(* check if inputs have chaged and fill buffer *)
IF s0 <> X0 THEN
	esr_out[cnt].typ := 10 + BOOL_TO_BYTE(s0);
	esr_out[cnt].adress := a0;
	esr_out[cnt].DS := DT_in;
	esr_out[cnt].TS := TX;
	X0 := S0;
	cnt := cnt + 1;
	esr_flag := TRUE;
END_IF;
IF s1 <> X1 THEN
	esr_out[cnt].typ := 10 + BOOL_TO_BYTE(s1);
	esr_out[cnt].adress := a1;
	esr_out[cnt].DS := DT_in;
	esr_out[cnt].TS := TX;
	X1 := S1;
	cnt := cnt + 1;
	esr_flag := TRUE;
END_IF;
IF s2 <> X2 THEN
	esr_out[cnt].typ := 10 + BOOL_TO_BYTE(s2);
	esr_out[cnt].adress := a2;
	esr_out[cnt].DS := DT_in;
	esr_out[cnt].TS := TX;
	X2 := S2;
	cnt := cnt + 1;
	esr_flag := TRUE;
END_IF;
IF s3 <> X3 THEN
	esr_out[cnt].typ := 10 + BOOL_TO_BYTE(s3);
	esr_out[cnt].adress := a3;
	esr_out[cnt].DS := DT_in;
	esr_out[cnt].TS := TX;
	X3 := S3;
	cnt := cnt + 1;
	esr_flag := TRUE;
END_IF;
IF s4 <> X4 AND cnt < 4 THEN
	esr_out[cnt].typ := 10 + BOOL_TO_BYTE(s4);
	esr_out[cnt].adress := a4;
	esr_out[cnt].DS := DT_in;
	esr_out[cnt].TS := TX;
	X4 := S4;
	cnt := cnt + 1;
	esr_flag := TRUE;
END_IF;
IF s5 <> X5  AND cnt < 4 THEN
	esr_out[cnt].typ := 10 + BOOL_TO_BYTE(s5);
	esr_out[cnt].adress := a5;
	esr_out[cnt].DS := DT_in;
	esr_out[cnt].TS := TX;
	X5 := S5;
	cnt := cnt + 1;
	esr_flag := TRUE;
END_IF;
IF s6 <> X6  AND cnt < 4 THEN
	esr_out[cnt].typ := 10 + BOOL_TO_BYTE(s6);
	esr_out[cnt].adress := a6;
	esr_out[cnt].DS := DT_in;
	esr_out[cnt].TS := TX;
	X6 := S6;
	cnt := cnt + 1;
	esr_flag := TRUE;
END_IF;
IF s7 <> X7  AND cnt < 4 THEN
	esr_out[cnt].typ := 10 + BOOL_TO_BYTE(s7);
	esr_out[cnt].adress := a7;
	esr_out[cnt].DS := DT_in;
	esr_out[cnt].TS := TX;
	X7 := S7;
	cnt := cnt + 1;
	esr_flag := TRUE;
END_IF;

(* revision history
hm	26. jan 2007	rev 1.0
	original version

hm	17. sep 2007	rev 1.1
	replaced time() with T_PLC_MS() for compatibility reasons

hm	22. oct. 2008	rev 1.2
	optimized code

hm	1.dec. 2009	rev 1.3
	changed esr_out to be I/O

*)
END_FUNCTION_BLOCK

(* POU Other/ESR_MON_R4, ST *)
FUNCTION_BLOCK ESR_MON_R4
VAR_INPUT
	R0, R1, R2, R3 : REAL;
	DT_in : DT;
END_VAR
VAR_INPUT CONSTANT
	a0, a1, a2, a3 : STRING(10);
	s0, s1, s2, s3 : REAL;
END_VAR
VAR_OUTPUT
	ESR_Flag : BOOL;
END_VAR
VAR_IN_OUT
	ESR_Out: ARRAY [0..3] OF esr_data;
END_VAR
VAR
	p0, p1, p2, p3 : POINTER TO DWORD;
	x0, x1, x2, x3 : REAL;
	tx: TIME;
	cnt : INT;
END_VAR

(*
version 1.4	1. dec. 2009
programmer 	hugo
tested by		tobias

ESR_mon_R4 monitores up to 4 Real inputs and reports changes with time stamd and adress label.
the module checks 4 inputs for a change of more than the specified sensitivity S and reports all changes with time and adress stamp to the output.

*)
(* read system timer *)
tx := DWORD_TO_TIME(T_PLC_MS());
P0 := ADR(R0);
P1 := ADR(R1);
P2 := ADR(R2);
P3 := ADR(R3);

ESR_Flag := FALSE;
esr_out[3].typ := 0;
esr_out[2].typ := 0;
esr_out[1].typ := 0;
esr_out[0].typ := 0;
cnt := 0;

(* check if inputs have chaged and fill buffer *)
IF DIFFER(R0,  X0, S0) THEN
	esr_out[cnt].typ := 20;
	esr_out[cnt].adress := a0;
	esr_out[cnt].DS := DT_in;
	esr_out[cnt].TS := TX;
	esr_out[cnt].data[0] := Byte_of_Dword(P0^,0);
	esr_out[cnt].data[1] := Byte_of_Dword(P0^,1);
	esr_out[cnt].data[2] := Byte_of_Dword(P0^,2);
	esr_out[cnt].data[3] := Byte_of_Dword(P0^,3);
	X0 := R0;
	cnt := cnt + 1;
	esr_flag := TRUE;
END_IF;
IF differ(R1,  X1, S1) THEN
	esr_out[cnt].typ := 20;
	esr_out[cnt].adress := a1;
	esr_out[cnt].DS := DT_in;
	esr_out[cnt].TS := TX;
	esr_out[cnt].data[0] := Byte_of_Dword(P1^,0);
	esr_out[cnt].data[1] := Byte_of_Dword(P1^,1);
	esr_out[cnt].data[2] := Byte_of_Dword(P1^,2);
	esr_out[cnt].data[3] := Byte_of_Dword(P1^,3);
	X1 := R1;
	cnt := cnt + 1;
	esr_flag := TRUE;
END_IF;
IF differ(R2,  X2, S2) THEN
	esr_out[cnt].typ := 20;
	esr_out[cnt].adress := a2;
	esr_out[cnt].DS := DT_in;
	esr_out[cnt].TS := TX;
	esr_out[cnt].data[0] := Byte_of_Dword(P2^,0);
	esr_out[cnt].data[1] := Byte_of_Dword(P2^,1);
	esr_out[cnt].data[2] := Byte_of_Dword(P2^,2);
	esr_out[cnt].data[3] := Byte_of_Dword(P2^,3);
	X2 := R2;
	cnt := cnt + 1;
	esr_flag := TRUE;
END_IF;
IF DIFFER(R3,  X3, S3) THEN
	esr_out[cnt].typ := 20;
	esr_out[cnt].adress := a3;
	esr_out[cnt].DS := DT_in;
	esr_out[cnt].TS := TX;
	esr_out[cnt].data[0] := Byte_of_Dword(P3^,0);
	esr_out[cnt].data[1] := Byte_of_Dword(P3^,1);
	esr_out[cnt].data[2] := Byte_of_Dword(P3^,2);
	esr_out[cnt].data[3] := Byte_of_Dword(P3^,3);
	X3 := R3;
	cnt := cnt + 1;
	esr_flag := TRUE;
END_IF;


(* revision history
hm	26. jan 2007	rev 1.0
	original version

hm	17. sep. 2007		rev 1.1
	replaced time() with T_PLC_MS() for compatibility reasons

hm	8. dec. 2007		rev 1.2
	corrected an error while esr typ would not be set

hm	16. mar. 2008		rev 1.3
	deleted wrong conversion real_to_dword

hm	1. dec 2009		rev 1.4
	changed esr_out to be I/O

*)
END_FUNCTION_BLOCK

(* POU Other/ESR_MON_X8, ST *)
FUNCTION_BLOCK ESR_MON_X8
VAR_INPUT
	s0, s1, s2, s3, s4, s5, s6, s7 : BYTE;
	DT_in : DT;
	Mode : BYTE := 3;
END_VAR
VAR_INPUT CONSTANT
	a0, a1, a2, a3, a4, a5, a6, a7 : STRING(10);
END_VAR
VAR_OUTPUT
	ESR_Flag : BOOL;
END_VAR
VAR_IN_OUT
	ESR_Out: ARRAY [0..3] OF esr_data;
END_VAR
VAR
	x0, x1, x2, x3, x4, x5, x6, x7 : BYTE;
	tx: TIME;
	cnt : INT;
END_VAR

(*
version 1.2	1. dec. 2009
programmer 	hugo
tested by		tobias

ESR_MON_X8 is a status and error collector.
the module checks 8 status inputs for a change and reports up to 4 input changes with time and adress stamp to the output.
the mode can be 
1 for error only
2 for error and status
3 for error, status and debug
the adress label of the 8 inputs can be configured individually.
*)
(* read system timer *)
tx := DWORD_TO_TIME(T_PLC_MS());

ESR_Flag := FALSE;
esr_out[3].typ := 0;
esr_out[2].typ := 0;
esr_out[1].typ := 0;
esr_out[0].typ := 0;
cnt := 0;


(* check if inputs have chaged and fill buffer *)
IF s0 <> X0 AND ((s0 < 100) OR (S0 > 99 AND S0 < 200 AND mode >= 2) OR (S0 > 199 AND mode = 3)) THEN
	esr_out[cnt] := status_to_ESR(s0, a0, DT_in, TX);
	X0 := S0;
	cnt := cnt + 1;
	esr_flag := TRUE;
END_IF;
IF s1 <> X1 AND ((s1 < 100) OR (S1 > 99 AND S1 < 200 AND mode >= 2) OR (S1 > 199 AND mode = 3)) THEN
	esr_out[cnt] := status_to_ESR(s1, a1, DT_in, TX);
	X1 := S1;
	cnt := cnt + 1;
	esr_flag := TRUE;
END_IF;
IF s2 <> X2 AND ((s2 < 100) OR (S2 > 99 AND S2 < 200 AND mode >= 2) OR (S2 > 199 AND mode = 3)) THEN
	esr_out[cnt] := status_to_ESR(s2, a2, DT_in, TX);
	X2 := S2;
	cnt := cnt + 1;
	esr_flag := TRUE;
END_IF;
IF s3 <> X3 AND ((s3 < 100) OR (S3 > 99 AND S3 < 200 AND mode >= 2) OR (S3 > 199 AND mode = 3)) THEN
	esr_out[cnt] := status_to_ESR(s3, a3, DT_in, TX);
	X3 := S3;
	cnt := cnt + 1;
	esr_flag := TRUE;
END_IF;
IF cnt < 4 AND s4 <> X4 AND ((s4 < 100) OR (S4 > 99 AND S4 < 200 AND mode >= 2) OR (S4 > 199 AND mode = 3)) THEN
	esr_out[cnt] := status_to_ESR(s4, a4, DT_in, TX);
	X4 := S4;
	cnt := cnt + 1;
	esr_flag := TRUE;
END_IF;
IF cnt < 4 AND s5 <> X5 AND ((s5 < 100) OR (S5 > 99 AND S5 < 200 AND mode >= 2) OR (S5 > 199 AND mode = 3)) THEN
	esr_out[cnt] := status_to_ESR(s5, a5, DT_in, TX);
	X5 := S5;
	cnt := cnt + 1;
	esr_flag := TRUE;
END_IF;
IF cnt < 4 AND s6 <> X6 AND ((s6 < 100) OR (S6 > 99 AND S6 < 200 AND mode >= 2) OR (S6 > 199 AND mode = 3)) THEN
	esr_out[cnt] := status_to_ESR(s6, a6, DT_in, TX);
	X6 := S6;
	cnt := cnt + 1;
	esr_flag := TRUE;
END_IF;
IF cnt < 4 AND s7 <> X7 AND ((s7 < 100) OR (S7 > 99 AND S7 < 200 AND mode >= 2) OR (S7 > 199 AND mode = 3)) THEN
	esr_out[cnt] := status_to_ESR(s7, a7, DT_in, TX);
	X7 := S7;
	cnt := cnt + 1;
	esr_flag := TRUE;
END_IF;


(* revision history
hm	26. jan 2007		rev 1.0
	original version

hm	17. sep 2007	rev 1.1
	replaced time() with T_PLC_MS() for compatibility reasons

hm	1. dec. 2009	rev 1.2
	changed esr_out to be I/O


*)
END_FUNCTION_BLOCK

(* POU Other/STATUS_TO_ESR, ST *)
FUNCTION STATUS_TO_ESR : esr_data
VAR_INPUT
	status : BYTE;
	adress : STRING(10);
	DT_in : DT;
	TS : TIME;
END_VAR


(*
version 1.0	6 oct 2006
programmer 	hugo
tested by		tobias

status_to_esr creates esr data from a status byte.

*)
IF status < 100 THEN
	status_to_ESR.typ := 1;
ELSIF status < 200 THEN
	status_to_ESR.typ := 2;
ELSE
	status_to_ESR.typ := 3;
END_IF;
status_to_ESR.adress:= adress;
status_to_ESR.DS := DT_in;
status_to_ESR.TS := TS;
status_to_ESR.data[0] := status;
END_FUNCTION

(* POU Other/OSCAT_VERSION, ST *)
FUNCTION OSCAT_VERSION : DWORD
VAR_INPUT
	IN : BOOL;
END_VAR


(*
version 1.1	16 dec 2007
programmer 	hugo
tested by		oscat

oscat_version returns the version number in dword format
132 is library version 1.32
if IN = true, the release date will be returned

*)
IF in THEN
	OSCAT_VERSION := DATE_TO_DWORD(D#2012-01-02);
ELSE
	OSCAT_VERSION := 333;
END_IF;

(* revision history
hm	6. oct 2006	rev 1.0
	original version

hm	16. dec 2007	rev 1.1
	added possibility to return date and version depending on IN.

*)
END_FUNCTION

(* POU String/BIN_TO_BYTE, ST *)
FUNCTION BIN_TO_BYTE : BYTE
VAR_INPUT
	BIN : STRING(12);
END_VAR
VAR
	pt : POINTER TO BYTE;
	i: INT;
	X: BYTE;
	stop: INT;
END_VAR

(*
version 1.2	26. jul 2009
programmer 	hugo
tested by		oscat

BINARY_TO_byte converts a binary string into a byte.

*)
pt := ADR(bin);
stop := LEN(bin);
FOR I := 1 TO stop DO
	x := pt^;
	(* calculate the value of the digit *)
	IF X = 48 THEN
		BIN_TO_BYTE := SHL(BIN_TO_BYTE,1);
	ELSIF X = 49 THEN
		BIN_TO_BYTE := SHL(BIN_TO_BYTE,1) OR 1;
	END_IF;
	pt := pt + 1;
END_FOR;



(* revision histroy
hm	18. jun. 2008	rev 1.0
	original release

hm	20. sep. 2008	rev 1.1
	changed length of input string from 20 to 12

hm	26. jul. 2009	rev 1.2
	optimized code
*)	
END_FUNCTION

(* POU String/BIN_TO_DWORD, ST *)
FUNCTION BIN_TO_DWORD : DWORD
VAR_INPUT
	BIN : STRING(40);
END_VAR
VAR
	pt : POINTER TO BYTE;
	i: INT;
	X: BYTE;
	stop: INT;
END_VAR

(*
version 1.2	26. jul. 2009
programmer 	hugo
tested by		oscat

BINARY_TO_DWORD converts a binary string into a dword.

*)
pt := ADR(bin);
stop := LEN(bin);
FOR I := 1 TO stop DO
	x := pt^;
	(* calculate the value of the digit *)
	IF X = 48 THEN
		BIN_TO_DWORD := SHL(BIN_TO_DWORD,1);
	ELSIF X = 49 THEN
		BIN_TO_DWORD := SHL(BIN_TO_DWORD,1) OR 1;
	END_IF;
	pt := pt + 1;
END_FOR;



(* revision histroy
hm	18. jun. 2008	rev 1.0
	original release

hm	20. sep. 2008	rev 1.1
	changed length of input dtring from 20 to 40

hm	26. jul 2009	rev 1.2
	optimized code
*)	
END_FUNCTION

(* POU String/BYTE_TO_STRB, ST *)
FUNCTION BYTE_TO_STRB : STRING(8)
VAR_INPUT
	IN : BYTE;
END_VAR
VAR
	i: INT;
	pt : POINTER TO BYTE;
END_VAR

(*
version 1.3	20. jun. 2008
programmer 	hugo
tested by	oscat

BYTE_TO_STRINGB converts a Byte to a String of Bits represented by '0' and '1' s.
The lowest order bit will be on the right and the high order bit on the left.

*)
(* pointer für die ausgabe ermitteln *)
pt := ADR(BYTE_TO_STRB);
(* die 8 ausgabecharacter ermitteln und schreiben *)
FOR i := 1 TO 8 DO
	pt^ := BOOL_TO_BYTE(in.7) + 48;
	in := SHL(in,1);
	pt := pt + 1;
END_FOR;

(* der ausgabestring muss noch mit 0 abgeschlossen werden *)
pt^ := 0;

(* code before rev 1.1
FOR i := 1 TO 8 DO
	IF in.0 = 0 THEN temp := CONCAT('0', temp); ELSE temp := CONCAT('1', temp); END_IF;
	in := SHR(in, 1);
END_FOR;
BYTE_TO_STRB := temp;
*)


(* revision history

hm		9.6.2007	rev 1.0		
	original version 

hm	15. dec 2007	rev 1.1
	inprooved code for higher performance

hm	29. mar. 2008	rev 1.2
	changed STRING to STRING(8)

hm	20. jun. 2008	rev 1.3
	performance improvement

*)
END_FUNCTION

(* POU String/BYTE_TO_STRH, ST *)
FUNCTION BYTE_TO_STRH : STRING(2)
VAR_INPUT
	IN : BYTE;
END_VAR
VAR
	temp : BYTE;
	PT : POINTER TO BYTE;
END_VAR

(*
version 1.3	29 mar. 2008
programmer 	hugo
tested by		tobias

BYTE_TO_STRINGH converts a Byte to a String of Hexadecimal represented by '0' .. '9' and 'A' .. 'F'.
The lowest order Character will be on the right and the high order Character on the left.

*)
(* read pointer to output string *)
PT := ADR(BYTE_TO_STRH);
(* calculate high order hex value *)
temp := SHR(in,4);
(* convert value to hex character *)
IF temp <= 9 THEN temp := temp + 48; ELSE temp := temp + 55; END_IF;
(* write friat character to output string *)
PT^ := temp;
(* calculate low order hex value *)
temp := in AND 2#00001111;
IF temp <= 9 THEN temp := temp + 48; ELSE temp := temp + 55; END_IF;
(* increment pointer and wirte low order character *)
pt := pt + 1;
pt^ := temp;
(* set pointer at the end of the output string and close the string with 0 *)
pt := pt + 1;
pt^:= 0;


(* code before rev 1.2
FOR i := 1 TO 2 DO
	X := in AND 2#1111;
	IF X <= 9 THEN X := X + 48; ELSE X := X + 55; END_IF;
	Cx := CHR(X);
	temp := CONCAT(Cx, temp);
	in := SHR(in,4);
END_FOR;
BYTE_TO_STRH := temp;
*)

(* revision history

hm	9.6.2007		rev 1.0		
	original version 

hm	11.9.2007		rev 1.1		
	changed coding for compatibility with twincat, under twincat concat cannot have a function as argument.	

hm	15 dec 2007		REV 1.2
	changed code for higher performance

hm	29. mar. 2008	rev 1.3
	changed STRING to STRING(2)
*)
END_FUNCTION

(* POU String/CAPITALIZE, ST *)
FUNCTION CAPITALIZE : STRING(STRING_LENGTH)
VAR_INPUT
	str : STRING(STRING_LENGTH);
END_VAR
VAR
	PT : POINTER TO BYTE;
	pos : INT;
	L : INT;
	first : BOOL := TRUE;
END_VAR

(*
version 1.2	20. jun. 2008
programmer 	hugo
tested by		tobias

capitalize returns str with all first letters after a blank or beginning of the string are converted to uppercase.

*)
PT := ADR(CAPITALIZE);
CAPITALIZE := str;
L := LEN(str);
FOR pos := 1 TO l DO
	IF first THEN pt^ := TO_UPPER(pt^);	END_IF;
	(* remember in first if the next char needs to capitalized *)
	first := pt^= 32;
	PT := pt + 1;
END_FOR;

(* revision histroy
hm		4. mar 2008	rev 1.0
	original release

hm	29. mar. 2008	rev 1.1
	changed STRING to STRING(STRING_LENGTH)

hm	20. jun. 2008	rev 1.2
	improved performance

*)	
END_FUNCTION

(* POU String/CHARCODE, ST *)
FUNCTION CHARCODE : BYTE
VAR_INPUT
	STR : STRING(10);
END_VAR
VAR
	found: STRING(1);
	search : STRING(10);
	pos: INT;
	i: INT;
END_VAR

(*
version 1.2		24. oct. 2008
programmer 		hugo
tested by		hugo

CHARCODE converts a HTML Character NAME INTO ITS code
'äuml' is convterted to ä
'euro' is converted to €

*)
IF LEN(str) = 1 THEN
	CHARCODE := CODE(STR, 1);
ELSIF str <> '' THEN
	(* construct search string *)
	search := CONCAT('&', str);
	search := CONCAT(search, ';');
	WHILE pos = 0 AND (i < 4) DO
		i := i + 1;
		pos := FIND(setup.CHARNAMES[i], search);
	END_WHILE;
	found := MID(setup.CHARNAMES[i], 1, pos - 1);
	CHARCODE := CODE(found, 1);
END_IF;




(* revision history
hm	13. may. 2008	rev 1.0
	original version

hm	19. oct. 2008	rev 1.1
	changed setup constants

hm	24. oct. 2008	rev 1.2
	optimized code
*)
END_FUNCTION

(* POU String/CHARNAME, ST *)
FUNCTION CHARNAME : STRING(10)
VAR_INPUT
	C : BYTE;
END_VAR
VAR
	pos: INT;
	i : INT;
END_VAR

(*
version 1.4		17. dec. 2008
programmer 		hugo
tested by		oscat

CHARNAME converts a Character code into its HTML character name
ä is convterted to 'äuml'
€ is converted to 'euro'
the character itself is returned if no name is available for the character

*)
IF C <> 0 THEN
	(* construct search string from code followed by $ sign, also clear charname string*)
	CHARNAME := CHR_TO_STRING(C);
	CHARNAME := CONCAT(CHARNAME,'&');
	CHARNAME := CONCAT(';', CHARNAME);
	WHILE pos = 0 AND (i < 4) DO
		i := i + 1;
		pos := FIND(setup.CHARNAMES[i], CHARNAME);
	END_WHILE;
	IF pos > 0 THEN
		CHARNAME := MID(setup.CHARNAMES[i], 10, pos + 3);
		(* search for end of name and truncate *)
		pos := FIND(CHARNAME, ';');
		CHARNAME := LEFT(CHARNAME,pos - 1);
	ELSE
		CHARNAME := CHR_TO_STRING(C);
	END_IF;
ELSE
	CHARNAME := '';
END_IF;




(* revision history
hm	13. may. 2008	rev 1.0
	original version

hm	16. jun. 2008	rev 1.1
	changed nested call of concat for better compatibility

hm	19. oct. 2008	rev 1.2
	changes setup constants

hm	24. oct. 2008	rev 1.3
	new code for high performance

hm	17. dec. 2008	rev 1.4
	changed function chr to chr_to_string
*)
END_FUNCTION

(* POU String/CLEAN, ST *)
FUNCTION CLEAN : STRING(STRING_LENGTH)
VAR_INPUT
	IN : STRING(STRING_LENGTH);
	CX : STRING(80);
END_VAR
VAR
	pos: INT := 1;
	stop: INT;
END_VAR


(*
version 1.0	18. jun. 2008
programmer 	hugo
tested by	oscat

Clean deletes all characters from a string except the ones specified in CX.

*)
(* copy input string *)
CLEAN := IN;
stop := LEN(in);
WHILE pos <= stop DO
	IF FIND(cx, MID(CLEAN, 1, pos)) > 0 THEN
		(* charcter found skip to next one *)
		pos := pos + 1;
	ELSE
		(* wrong chracter needs to be deleted *)
		CLEAN := DELETE(CLEAN, 1, pos);
		stop := stop - 1;	(* the string is one character shorter now *)
	END_IF;
END_WHILE;



(* revision history

hm		18. jun. 2008	rev 1.0		
	original version 


*)
END_FUNCTION

(* POU String/COUNT_CHAR, ST *)
FUNCTION COUNT_CHAR : INT
VAR_INPUT
	str : STRING(STRING_LENGTH);
	chr : BYTE;
END_VAR
VAR
	l: INT;
	pt : POINTER TO BYTE;
	pos: INT;
END_VAR


(*
version 1.1	29. mar. 2008
programmer 		kurt
tested by		hugo

COUNT_CHAR counts how often a character CHAR occurs within a string STR.

*)
PT := ADR(str);
l := LEN(str);
COUNT_CHAR := 0;
FOR pos := 1 TO l DO
	IF pt^ = CHR THEN COUNT_CHAR := COUNT_CHAR + 1; END_IF;
    PT := PT + 1;
END_FOR;


(* revision history
hm	29. feb 2008	rev 1.0
	original version

hm	29. mar. 2008	rev 1.1
	changed STRING to STRING(STRING_LENGTH)
*)
END_FUNCTION

(* POU String/COUNT_SUBSTRING, ST *)
FUNCTION COUNT_SUBSTRING : INT
VAR_INPUT
   SEARCH : STRING;
   STR : STRING;
END_VAR
VAR
   pos : INT;
   size : INT;
END_VAR

(*
version 1.0	20. jan. 2011
programmed	kurt
tested by		tobias

count_substring returns the number of occurences of a substring in a string

*)
COUNT_SUBSTRING := 0;
size := LEN(SEARCH);
REPEAT
   pos := FIND(STR,SEARCH);
   IF pos > 0 THEN
      STR := REPLACE(STR, '', size,pos);
      COUNT_SUBSTRING := COUNT_SUBSTRING + 1;
   END_IF;
UNTIL pos = 0
END_REPEAT;


(* revision history
ks	20. jan. 2011	rev 1.0
	original version

*)
END_FUNCTION

(* POU String/DEC_TO_BYTE, ST *)
FUNCTION DEC_TO_BYTE : BYTE
VAR_INPUT
	DEC : STRING(10);
END_VAR
VAR
	pt : POINTER TO BYTE;
	i: INT;
	X: BYTE;
	stop: INT;
END_VAR

(*
version 1.1	30. sep 2008
programmer 	hugo
tested by		oscat

DEC_TO_byte converts a decimal string into a byte.

*)
pt := ADR(dec);
stop := LEN(DEC);
FOR I := 1 TO stop DO
	(* read the first character and subtract 48 to get value in decimal 0 = 48 *)
	x := pt^;
	(* calculate the value of the digit *)
	IF X > 47 AND x < 58 THEN
		DEC_TO_BYTE := DEC_TO_BYTE * 10 + X - 48;
	END_IF;
	pt := pt + 1;
END_FOR;



(* revision histroy
hm	20. jun. 2008	rev 1.0
	original release

hm	30. sep.2008	rev 1.1
	changed length of input string from 20 to 10
	corrected an error where decoding of characters 8 and 9 would fail

*)	
END_FUNCTION

(* POU String/DEC_TO_DWORD, ST *)
FUNCTION DEC_TO_DWORD : DWORD
VAR_INPUT
	DEC : STRING(20);
END_VAR
VAR
	pt : POINTER TO BYTE;
	i: INT;
	X: BYTE;
	stop: INT;
END_VAR

(*
version 1.1	30. sep. 2008
programmer 	hugo
tested by		oscat

DEC_TO_DWORD converts a decimal string into a DWORD.

*)
pt := ADR(dec);
stop := LEN(dec);
FOR I := 1 TO stop DO
	(* read the first character and subtract 48 to get value in decimal 0 = 48 *)
	x := pt^;
	(* calculate the value of the digit *)
	IF X > 47 AND x < 58 THEN
		DEC_TO_DWORD := DEC_TO_DWORD * 10 + X - 48;
	END_IF;
	pt := pt + 1;
END_FOR;



(* revision histroy
hm	20. jun. 2008	rev 1.0
	original release

hm	30. sep. 2008	rev 1.1
	corrected an error where decoding of characters 8 and 9 would fail
*)	
END_FUNCTION

(* POU String/DEC_TO_INT, ST *)
FUNCTION DEC_TO_INT : INT
VAR_INPUT
	DEC : STRING(10);
END_VAR
VAR
	pt : POINTER TO BYTE;
	i: INT;
	X: BYTE;
	sign: BOOL;
	stop: INT;
END_VAR

(*
version 1.1	30. sep. 2008
programmer 	hugo
tested by	oscat

DEC_TO_INT converts a decimal string into an Integer.

*)
pt := ADR(dec);
stop := LEN(dec);
FOR I := 1 TO stop DO
	(* read the first character and subtract 48 to get value in decimal 0 = 48 *)
	x := pt^;
	(* calculate the value of the digit *)
	IF X > 47 AND x < 58 THEN
		DEC_TO_INT := DEC_TO_INT * 10 + X - 48;
	ELSIF X = 45 AND DEC_TO_INT = 0 THEN
		sign := TRUE;
	END_IF;
	pt := pt + 1;
END_FOR;
IF sign THEN DEC_TO_INT := -DEC_TO_INT; END_IF;


(* revision histroy
hm	20. jun. 2008	rev 1.0
	original release

hm	30. sep. 2008	rev 1.1
	changed length of input string from 20 to 10
	corrected an error where decoding of characters 8 and 9 would fail
*)	
END_FUNCTION

(* POU String/DEL_CHARS, ST *)
FUNCTION DEL_CHARS : STRING(STRING_LENGTH)
VAR_INPUT
	IN : STRING(STRING_LENGTH);
	CX : STRING(80);
END_VAR
VAR
	pos: INT := 1;
	stop: INT;
END_VAR


(*
version 1.0	18. jun. 2008
programmer 	hugo
tested by	oscat

del_chars deletes all characters from a string which are specified in CX.

*)
(* copy input string *)
DEL_CHARS := IN;
stop := LEN(in);
WHILE pos <= stop DO
	IF FIND(cx, MID(DEL_CHARS, 1, pos)) > 0 THEN
		(* wrong chracter needs to be deleted *)
		DEL_CHARS := DELETE(DEL_CHARS, 1, pos);
		stop := stop - 1;	(* the string is one character shorter now *)
	ELSE
		(* charcter not found skip to next one *)
		pos := pos + 1;
	END_IF;
END_WHILE;



(* revision history

hm		18. jun. 2008	rev 1.0		
	original version 


*)
END_FUNCTION

(* POU String/DT_TO_STRF, ST *)
FUNCTION DT_TO_STRF : STRING
VAR_INPUT
	DTI : DT;
	MS : INT;
	FMT : STRING;
	LANG : INT;
END_VAR
VAR CONSTANT
	FILL : STRING(1) := '0';
	BLANK : STRING(1) := ' ';
END_VAR
VAR
	ly : INT;
	dx: DATE;
	fs: STRING(10);
	td: TOD;
	tmp : INT;
	pos : INT;
	f : INT;
END_VAR

(*
version 1.1	19. oct. 2008
programmer 	hugo
tested by	oscat

DT_TO_STRINGF converts a DATETIME input to a formatted string

*)
IF LANG < 1 THEN ly := language.DEFAULT; ELSE ly := MIN(language.LMAX, LANG); END_IF;

(* decode date and time information *)
dx := DT_TO_DATE(DTI);
td := DT_TO_TOD(DTI);

(* parse the format string *)
DT_TO_STRF := FMT;
pos := FIND(DT_TO_STRF, '#');
WHILE pos > 0 DO
	(* retrieve format identifier *)
	f := CODE(DT_TO_STRF, pos + 1);
	(* generate the return string according to the format character *)
	fs := '';
	CASE f OF
		65 : (* letter A retunrs the year in 4 digits *)
			fs := INT_TO_STRING(YEAR_OF_DATE(dx));
		66 : (* letter B returns the year in exactly 2 digits *)
			fs := RIGHT(INT_TO_STRING(YEAR_OF_DATE(dx)),2);
		67 : (* letter C returns the month with 1 or 2 digits *)
			fs := INT_TO_STRING(MONTH_OF_DATE(dx));
		68 : (* letter D returns the month with exactly 2 digits *)
			fs := INT_TO_STRING(MONTH_OF_DATE(dx));
			IF LEN(fs) < 2 THEN fs := CONCAT('0', fs); END_IF;
		69 : (* letter E returns the month with 3 characters *)
			fs := MONTH_TO_STRING(MONTH_OF_DATE(dx), ly, 3);
		70 : (* letter F returns the month with all characters *)
			fs := MONTH_TO_STRING(MONTH_OF_DATE(dx), ly, 0);
		71 : (* letter G returns the day with up to 2 digits *)
			fs := INT_TO_STRING(DAY_OF_MONTH(dx));
		72 : (* letter H returns the day of the month with exactly 2 digits *)
			fs := INT_TO_STRING(DAY_OF_MONTH(dx));
			IF LEN(fs) < 2 THEN fs := CONCAT(FILL, fs); END_IF;
		73 : (* letter I returns the weekday as the number 1..7 1 = monday *)
			fs := INT_TO_STRING(DAY_OF_WEEK(dx));
		74 : (* letter J returns the weekday in 2 character writing *)
			fs := WEEKDAY_TO_STRING(DAY_OF_WEEK(dx), ly, 2);
		75 : (* letter K returns the weekday with all characters *)
			fs := WEEKDAY_TO_STRING(DAY_OF_WEEK(dx), ly, 0);
		76 : (* letter L returns AM or PM for the given DateTime *)
			IF td >= TOD#12:00 THEN fs := 'PM'; ELSE fs := 'AM'; END_IF;
		77 : (* letter M returns the hour in 1 or 2 digit form 0..24h *)
			fs := INT_TO_STRING(HOUR(td));
		78 : (* letter N returns the hour in exactly 2 digit form 0..24h *)
			fs := INT_TO_STRING(HOUR(td));
			IF LEN(fs) < 2 THEN fs := CONCAT(FILL, fs); END_IF;
		79 : (* letter O returns the hour in 1 or 2 digit form 0..12h *)
			tmp := HOUR(td) MOD 12;
			IF tmp = 0 THEN tmp := 12; END_IF;
			fs := INT_TO_STRING(tmp);
		80 : (* letter P returns the hour in exactly 2 digit form 0..12h *)
			tmp := HOUR(td) MOD 12;
			IF tmp = 0 THEN tmp := 12; END_IF;
			fs := INT_TO_STRING(tmp);
			IF LEN(fs) < 2 THEN fs := CONCAT(FILL, fs); END_IF;
		81 : (* letter Q returns the minute of the hour in 1 or two digit form *)
			fs := INT_TO_STRING(MINUTE(td));
		82 : (* letter R returns the minute of the hour in exactly two digit form *)
			fs := INT_TO_STRING(MINUTE(td));
			IF LEN(fs) < 2 THEN fs := CONCAT(FILL, fs); END_IF;
		83 : (* letter S returns the second of the minute in 1 or two digit form *)
			fs := INT_TO_STRING(REAL_TO_INT(SECOND(td)));
		84 : (* letter T returns the second of the minute in exactly two digit form *)
			fs := INT_TO_STRING(REAL_TO_INT(SECOND(td)));
			IF LEN(fs) < 2 THEN fs := CONCAT(FILL, fs); END_IF;
		85 : (* letter U returns the milliseconds in 1 to 3 digits *)
			fs := INT_TO_STRING(MS);
		86 : (* letter V returns the milliseconds in exactly 3 digit form *)
			fs := INT_TO_STRING(MS);
			fs := CONCAT('00',fs);
			fs := RIGHT(fs, 3);
		87 : (* letter W returns the day of the month with exactly 2 digits first digit is filled with blank if necessary *)
			fs := INT_TO_STRING(DAY_OF_MONTH(dx));
			IF LEN(fs) < 2 THEN fs := CONCAT(BLANK, fs); END_IF;
		88 : (* letter X returns the month with exactly 2 digits first digit is filled with blank if necessary *)
			fs := INT_TO_STRING(MONTH_OF_DATE(dx));
			IF LEN(fs) < 2 THEN fs := CONCAT(BLANK, fs); END_IF;
		END_CASE;
	DT_TO_STRF := REPLACE(DT_TO_STRF, fs, 2, pos);
	pos := FIND(DT_TO_STRF, '#');
END_WHILE;


(* revision history
hm	7. oct. 2008	rev 1.0
	original version

hm	19. oct. 2008	rev 1.1
	changed language setup constants
*)
END_FUNCTION

(* POU String/FILL, ST *)
FUNCTION FILL : STRING(STRING_LENGTH)
VAR_INPUT
	C : BYTE;
	L : INT;
END_VAR
VAR
	i: INT;
	sx: STRING(1);
END_VAR

(*
version 1.1	17. dec. 2008
programmer 	hugo
tested by		tobias

the function fill creates a string at length L of characters C.

*)
Sx := CHR_TO_STRING(c);
(* limit L to maximum 80 characters the length of a standard string *)
L := LIMIT(0,L,STRING_LENGTH);
(* create a string of characters to be connected to str *)
FOR i := 1 TO 8 DO
	FILL := CONCAT(FILL,FILL);
	IF L.7 THEN FILL := CONCAT(FILL,Sx); END_IF;
	L := SHL(L,1);
END_FOR;




(* revision histroy
hm	29. mar. 2008	rev 1.0
	original release

hm	17. dec. 2008	rev 1.1
	changed function chr to chr_to_string

*)
END_FUNCTION

(* POU String/MONTH_TO_STRING, ST *)
FUNCTION MONTH_TO_STRING : STRING(10)
VAR_INPUT
	MTH : INT;
	LANG : INT;
	LX : INT;
END_VAR
VAR
	ly : INT;
END_VAR

(*
version 1.1	19. oct. 2008
programmer 	hugo
tested by	oscat

MONTH_TO_STRING converts an Integer 1..12 into a String with the Names of the corresponding Month.
the decoding is according to the language setup in global vars

*)
IF LANG = 0 THEN Ly := LANGUAGE.DEFAULT; ELSE ly := MIN(LANG, language.LMAX); END_IF;
IF MTH < 1 OR MTH > 12 THEN
	RETURN;
ELSIF LX = 0 THEN
	MONTH_TO_STRING := language.MONTHS[ly, MTH];
ELSIF Lx = 3 THEN
	MONTH_TO_STRING := language.MONTHS3[ly, MTH];
END_IF;


(* revisison history

hm	21. sep. 2008	rev 1.0
	original version

hm	19. oct. 2008	rev 1.1
	changed language setup constants
*)
END_FUNCTION

(* POU Time&Date/DAY_OF_MONTH, ST *)
FUNCTION DAY_OF_MONTH : INT
VAR_INPUT
	IDATE : DATE;
END_VAR
VAR
	leap: INT;
END_VAR

(*
version 2.1	10. mar. 2009
programmer 	hugo
tested by		tobias

returns the day OF month for any DATE

*)
(* calculate the day in the year *)
DAY_OF_MONTH := DAY_OF_YEAR(idate);
(* leap will be set to one for a leap year *)
leap := BOOL_TO_INT(LEAP_OF_DATE(idate));
(* if leap year deduct one from the days of the year *)
DAY_OF_MONTH := DAY_OF_MONTH - leap;
(* search if we are in month december to march ? *)
IF DAY_OF_MONTH > setup.MTH_OFS[9] THEN
	IF DAY_OF_MONTH > setup.MTH_OFS[11] THEN
		IF DAY_OF_MONTH > setup.mth_ofs[12] THEN
			DAY_OF_MONTH := DAY_OF_MONTH - setup.MTH_OFS[12];
		ELSE
			DAY_OF_MONTH := DAY_OF_MONTH - setup.MTH_OFS[11];
		END_IF;
	ELSE
		IF DAY_OF_MONTH > setup.mth_ofs[10] THEN
			DAY_OF_MONTH := DAY_OF_MONTH - setup.MTH_OFS[10];
		ELSE
			DAY_OF_MONTH := DAY_OF_MONTH - setup.MTH_OFS[9];
		END_IF;
	END_IF;
ELSIF DAY_OF_MONTH > setup.MTH_OFS[5] THEN
	IF DAY_OF_MONTH > setup.MTH_OFS[7] THEN
		IF DAY_OF_MONTH > setup.mth_ofs[8] THEN
			DAY_OF_MONTH := DAY_OF_MONTH - setup.MTH_OFS[8];
		ELSE
			DAY_OF_MONTH := DAY_OF_MONTH - setup.MTH_OFS[7];
		END_IF;
	ELSE
		IF DAY_OF_MONTH > setup.mth_ofs[6] THEN
			DAY_OF_MONTH := DAY_OF_MONTH - setup.MTH_OFS[6];
		ELSE
			DAY_OF_MONTH := DAY_OF_MONTH - setup.MTH_OFS[5];
		END_IF;
	END_IF;
ELSIF DAY_OF_MONTH > setup.MTH_OFS[3] THEN
	IF DAY_OF_MONTH > setup.MTH_OFS[4] THEN
		DAY_OF_MONTH := DAY_OF_MONTH - setup.MTH_OFS[4];
	ELSE
		DAY_OF_MONTH := DAY_OF_MONTH - setup.MTH_OFS[3];
	END_IF;
ELSE
	(* since now we must be in february or january we need to add leap again *)
	DAY_OF_MONTH := DAY_OF_MONTH + leap;
	IF DAY_OF_MONTH > setup.MTH_OFS[2] THEN DAY_OF_MONTH := DAY_OF_MONTH - setup.mth_ofs[2]; END_IF;
	(* since nothing was true before, day_of_month must already be good *)
END_IF;


(*
Revision history

hm 22.1.2007		rev 1.1
	deleted unused variable day_in_year and day_in_year_begin

hm	1. okt 2007	rev 1.2
	changed code to use day_of_year and leap_of_date
	added compatibility to STEP7

hm	8. oct 2007	rev 1.3
	deleted unused variable yr

hm	8. jan 2008	rev 1.4
	improved performance

hm	25. oct. 2008	rev 2.0
	new code using setup constants

hm	10. mar. 2009	rev 2.1
	removed nested comments

*)
END_FUNCTION

(* POU String/WEEKDAY_TO_STRING, ST *)
FUNCTION WEEKDAY_TO_STRING : STRING(10)
VAR_INPUT
	WDAY : INT;
	LANG : INT;
	LX : INT;
END_VAR
VAR
	ly : INT;
END_VAR

(*
version 1.1	19. oct. 2008
programmer 	hugo
tested by	oscat

WEEKDAY_TO_STRING converts an Integer 1..7 into a String with the Names of the corresponding weekday.
the decoding is according to the language setup in global vars

*)
IF LANG = 0 THEN ly := LANGUAGE.DEFAULT; ELSE ly := MIN(LANG, LANGUAGE.LMAX); END_IF;
IF wday < 1 OR wday > 7 THEN
	RETURN;
ELSIF LX = 0 THEN
	WEEKDAY_TO_STRING := language.WEEKDAYS[ly, WDAY];
ELSIF Lx = 2 THEN
	WEEKDAY_TO_STRING := language.WEEKDAYS2[ly, WDAY];
END_IF;


(* revisison history

hm	21. sep. 2008	rev 1.0
	original version

hm	19. oct. 2008	rev 1.1
	changed language setup constants
*)
END_FUNCTION

(* POU Time&Date/HOUR, ST *)
FUNCTION HOUR : INT
VAR_INPUT
	itod : TOD;
END_VAR


(*
version 1.1	2 okt 2006
programmer 	hugo
tested by	tobias

extracts the hour of a Time_of_day 
*)
HOUR := DWORD_TO_INT(TOD_TO_DWORD(itod) / 3600000);


(* change history
hm 4. aug 2006	rev 1.0
	original version

hm 2.10.2006 	rev 1.1
	changed name of input to itod

*)
END_FUNCTION

(* POU Time&Date/MINUTE, ST *)
FUNCTION MINUTE : INT
VAR_INPUT
	itod : TOD;
END_VAR


(*
version 1.1	2 oct 2006
programmer 	hugo
tested by	tobias

extracts the minutes out of TOD truncating the seconds 

*)  
MINUTE := DWORD_TO_INT(TOD_TO_DWORD(itod) / 60000 - TOD_TO_DWORD(itod) / 3600000 * 60);


(* change history

2.10.2006 changes name of input to itod

*)
END_FUNCTION

(* POU Time&Date/SECOND, ST *)
FUNCTION SECOND : REAL
VAR_INPUT
	itod : TOD;
END_VAR


(*
version 1.1	2 oct 2006
programmer 	hugo
tested by	oscat

returns the seconds and milliseconds as real of TOD   
 
*)
SECOND := DWORD_TO_REAL(TOD_TO_DWORD(itod) - TOD_TO_DWORD(itod)/60000 * 60000) / 1000.0;



(* change history

hm	2. oct. 2006 rev 1.1 
	changed name of input to itod

*)
END_FUNCTION

(* POU String/DWORD_TO_STRB, ST *)
FUNCTION DWORD_TO_STRB : STRING(32)
VAR_INPUT
	IN : DWORD;
END_VAR
VAR
	pt : POINTER TO BYTE;
	i: INT;
END_VAR

(*
version 1.3	20. jun. 2008
programmer 	hugo
tested by	oscat

DWORD_TO_STRINGB converts a DWORD to a String of Bits represented by '0' and '1' s.
The lowest order bit will be on the right and the high order bit on the left.

*)
(* pointer für die ausgabe ermitteln *)
pt := ADR(DWORD_TO_STRB);
(* die 8 ausgabecharacter ermitteln und schreiben *)
FOR i := 1 TO 32 DO
	pt^:= BOOL_TO_BYTE(in.31) + 48;
	in := SHL(in,1);
	pt := pt + 1;
END_FOR;

(* der ausgabestring muss nochg mit 0 abgeschlossen werden *)
pt^ := 0;

(* revision history
hm		9.6.2007	rev 1.0		
	original version

hm		15.dec 2007	rev 1.1
	changed code for better performance

hm	29. mar. 2008	rev 1.2
	changed STRING to STRING(32)

hm	20. jun. 2008	rev 1.3
	performance improvement

*)
END_FUNCTION

(* POU String/DWORD_TO_STRF, ST *)
FUNCTION DWORD_TO_STRF : STRING(20)
VAR_INPUT
	IN : DWORD;
	N : INT;
END_VAR


(*
version 1.0	26 jan 2007
programmer 	hugo
tested by		tobias

dword_to_strF converts a DWORD, BYTE or Word to a fixed length String.
the string will be filled with leading zeroes to achieve the fixed length, or if too long, the lowest digits will be used.
the maximum allowed length is 20 mdigits.

for example:	dword_to_strf(123,4) = '0123' 
				dword_to_strf(123,2) = '23'
*)
(* limit N to max 20 characters *)
(* convert dword to string first and cut to length N *)
DWORD_TO_STRF := FIX(DWORD_TO_STRING(in),LIMIT(0,N,20),48,1);


(* revision history
hm	26. jan.2007	rev 1.0		
	original version

hm	29. mar. 2008	rev 1.1
	changed STRING to STRING(20)
	limit the output string to max 20 digits
*)
END_FUNCTION

(* POU String/FIX, ST *)
FUNCTION FIX : STRING(STRING_LENGTH)
VAR_INPUT
	str : STRING(STRING_LENGTH);
	L : INT;
	C : BYTE;
	M : INT;
END_VAR
VAR
	N : INT;
	SX: STRING(STRING_LENGTH);
END_VAR

(*
version 1.0	29. mar. 2008
programmer 	hugo
tested by	tobias

the function fix truncates a string at length L 
or if the string is shorter then L it will be filled with ending Spaces till its length = N.

*)
(* make sure L does not exceed the limits of a string *)
N := LIMIT(0,L,STRING_LENGTH) - LEN(str);
IF N <= 0 THEN
	(* truncate the string at length N *)
	IF M = 1 THEN
		FIX := RIGHT(str,L);
	ELSE
		FIX := LEFT(str,L);
	END_IF;
ELSIF M = 1 THEN
	(* connect fill characters at the beginning *)
	sx := FILL(C,N);
	FIX := CONCAT(sx,str);
ELSIF M = 2 THEN
	(* center str beween fill characters *)
	(* for an uneven number of fill characters, there is one more at the end *)
	sx := FILL(C,SHR(N+1,1));
	FIX := CONCAT(str,sx);
	SX := LEFT(sx,SHR(N,1));
	FIX := CONCAT(sx,FIX);
ELSE
	(* connect fill characters at the end *)
	SX := FILL(C,N);
	FIX := CONCAT(str,SX);
END_IF;


(* revision histroy
hm	29. mar. 2008	rev 1.0
	original release

*)
END_FUNCTION

(* POU String/DWORD_TO_STRH, ST *)
FUNCTION DWORD_TO_STRH : STRING(8)
VAR_INPUT
	IN : DWORD;
END_VAR
VAR
	i : INT;
	temp : BYTE;
	pt : POINTER TO BYTE;
END_VAR

(*
version 1.3	29. mar. 2008
programmer 	hugo
tested by	tobias

DWORD_TO_STRINGH converts a DWORD to a String of Hexadecimal represented by '0' .. '9' and 'A' .. 'F'.
The lowest order Character will be on the right and the high order Character on the left.

*)
(* read output adress to pointer *)
pt := ADR(DWORD_TO_STRH) + 8;
(* wirte the closing byte for the string *)
pt^:= 0;

(* write the 8 hex characters backwards *)
FOR i := 1 TO 8 DO;
	(* decrement the pointer *)
	pt := pt - 1;
	(* read the lowest order hex value *)
	temp := DWORD_TO_BYTE(in AND 16#0000000F);
	(* convert value to hex character *)
	IF temp <= 9 THEN temp := temp + 48; ELSE temp := temp + 55; END_IF;
	(* write character to output string *)
	PT^ := temp;
	(* shift in for nect hex character *)
	in := SHR(in,4);
END_FOR;


(* code beofre rev 1.2
FOR i := 1 TO 8 DO
	X := DWORD_TO_BYTE(in AND 2#1111);
	IF X <= 9 THEN X := X + 48; ELSE X := X + 55; END_IF;
	Cx := CHR(X);
	temp := CONCAT(Cx, temp);
	in := SHR(in,4);
END_FOR;
DWORD_TO_STRH := temp;
*)


(* revision history
hm	9. jun. 2007	rev 1.0		
	original version 

hm	11. sep. 2007	rev 1.1
	changed coding for compatibility with twincat, concat cannot support a function as an argument.

hm	15. dec. 2007	rev 1.2
	changed code for better performance

hm	29. mar. 2008	rev 1.3
	changed STRING to STRING(8)

*)
END_FUNCTION

(* POU String/EXEC, ST *)
FUNCTION EXEC : STRING(STRING_LENGTH)
VAR_INPUT
	str : STRING(STRING_LENGTH);
END_VAR
VAR
	pos: INT;
	R1: REAL;
	R2: REAL;
	operator: STRING(10);
END_VAR

(*
version 1.4	29. mar. 2008
programmer 	hugo
tested by		tobias

exec executes a mathematical term and returns the result as a string
the term can only be a simple term without brackets and only one operator
allowed operastors are: (+, -, *, /, ^, sqrt, sin, cos, tan).

*)
(* extract both numbers and operator *)
EXEC := UPPERCASE(TRIM(str));

pos := FINDB_NONUM(EXEC);
IF pos > 1 THEN R1 := STRING_TO_REAL(LEFT(EXEC,pos-1)); END_IF;
R2 := STRING_TO_REAL(RIGHT(EXEC,LEN(EXEC)-pos));
EXEC := LEFT(EXEC,pos);
pos := FINDB_NUM(EXEC);
operator := RIGHT(EXEC,LEN(EXEC) - pos);
IF operator = '' AND LEN(str) = 0 THEN
	EXEC := '';
	RETURN;
ELSIF operator = '' THEN
	EXEC := str;
	RETURN;
END_IF;
IF operator = '^' THEN
	EXEC := REAL_TO_STRING(EXPT(R1, R2));
ELSIF operator = 'SQRT' THEN
	EXEC := REAL_TO_STRING(SQRT(R2));
ELSIF operator = 'SIN' THEN
	EXEC := REAL_TO_STRING(SIN(r2));
ELSIF operator = 'COS' THEN
	EXEC := REAL_TO_STRING(COS(r2));
ELSIF operator = 'TAN' THEN
	EXEC := REAL_TO_STRING(TAN(R2));
ELSIF operator = '*' THEN
	EXEC := REAL_TO_STRING(R1 * R2);
ELSIF operator = '/' THEN
	IF R2 <> 0 THEN EXEC := REAL_TO_STRING(R1 / R2); ELSE EXEC := 'ERROR'; END_IF;
ELSIF operator = '+' THEN
	EXEC := REAL_TO_STRING(r1 + r2);
ELSIF operator = '-' THEN
	EXEC := REAL_TO_STRING(r1 - r2);
ELSE
	EXEC := 'ERROR';
END_IF;

IF EXEC = 'ERROR' THEN
	RETURN;
(* some systems deliver integer instead of real *)
ELSIF FIND(EXEC,'.') = 0 THEN
	EXEC := CONCAT(EXEC, '.0');
(* some systems deliver n. instead of n.0 ! *)
ELSIF RIGHT(EXEC,1) = '.' THEN
	EXEC := CONCAT(EXEC,'0');
END_IF;


(* revision history

hm 	6.feb 2007		rev 1.1
	cos has to be written in uppercase
	divide by 0 will return an error

hm	5. mar. 2008	rev 1.2
	add a 0 to the string if a '.' is at the end of the string

hm	20. mar. 2008	rev 1.3
	make sure the function always returns a real value in the form of x.y

hm	29. mar. 2008	rev 1.4
	changed STRING to STRING(STRING_LENGTH)
*)
END_FUNCTION

(* POU String/UPPERCASE, ST *)
FUNCTION UPPERCASE : STRING(STRING_LENGTH)
VAR_INPUT
	str : STRING(STRING_LENGTH);
END_VAR
VAR
	pt : POINTER TO BYTE;
	pos: INT;
	l: INT;
END_VAR

(*
version 1.3	29. mar. 2008
programmer 	hugo
tested by	tobias

uppercase returns str while all letters a..z and ä,ö,ü are converted to uppercase

*)
pt := ADR(UPPERCASE);
UPPERCASE := str;
l := LEN(str);
FOR pos := 1 TO l DO
	pt^ := TO_UPPER(pt^);
	pt := pt + 1;
END_FOR;

(* revision histroy
hm	6. oct. 2006	rev 1.0
	original release

hm	4. feb. 2008	rev 1.1
	improved performance
	added Ä,Ö,Ü

hm	6. mar. 2008	rev 1.2
	added support for exteded Ascii

hm	29. mar. 2008	rev 1.3
	changed STRING to STRING(STRING_LENGTH)

*)	
END_FUNCTION

(* POU String/TRIM, ST *)
FUNCTION TRIM : STRING(STRING_LENGTH)
VAR_INPUT
	str : STRING(STRING_LENGTH);
END_VAR
VAR
	pos: INT;
END_VAR

(*
version 1.2	29. mar. 2008
programmer 	hugo
tested by	tobias

the function deletes all blanks within a string.

*)
TRIM := str;
REPEAT
	pos := FIND(trim,' ');
	IF pos > 0 THEN TRIM := REPLACE(TRIM,'',1,pos); END_IF;
UNTIL pos = 0	END_REPEAT;


(* revision histroy
hm	6.10.2006		rev 1.0
	original release

hm	20. mar. 2008	rev 1.1
	avoid to call replace with pos = 0 because some systems will produce an error

hm	29. mar. 2008	rev 1.2
	changed STRING to STRING(STRING_LENGTH)
*)
END_FUNCTION

(* POU String/FINDB_NONUM, ST *)
FUNCTION FINDB_NONUM : INT
VAR_INPUT
	str : STRING(STRING_LENGTH);
END_VAR
VAR
	pos: INT;
	pt : POINTER TO BYTE;
END_VAR

(*
version 1.3	21. oct. 2008
programmer 	hugo
tested by	oscat

findB_noNum searches str backwards and returns the last position which is not a number.
a number is characterized by a letter "0..9" or "."

*)
pt := ADR(str) + LEN(str) - 1;
FOR pos := LEN(str) TO 1 BY -1 DO;
	IF (PT^ < 48 AND PT^ <> 46) OR PT^ > 57 THEN
		FINDB_NONUM := pos;
		RETURN;
	END_IF;
	PT := PT - 1;
END_FOR;
FINDB_NONUM := 0;


(* revision history
hm	6. oct 2006		rev 1.0
	original version

hm	29. feb 2008	rev 1.1
	improved performance

hm	29. mar. 2008	rev 1.2
	changed STRING to STRING(STRING_LENGTH)

hm	21. oct. 2008	rev 1.3
	optimized code
*)
END_FUNCTION

(* POU String/FINDB_NUM, ST *)
FUNCTION FINDB_NUM : INT
VAR_INPUT
	str : STRING(STRING_LENGTH);
END_VAR
VAR
	pos: INT;
	pt : POINTER TO BYTE;
END_VAR

(*
version 1.2	29. mar. 2008
programmer 	hugo
tested by	tobias

findB_Num searches str backward and returns the last position of a number
a number is characterized by a letter "0..9" or "."

*)
pt := ADR(str) + LEN(str) - 1;
FOR pos := LEN(str) TO 1 BY -1 DO;
	IF (PT^ > 47 AND PT^ < 58) OR PT^ = 46 THEN
		FINDB_NUM := pos;
		RETURN;
	END_IF;
	PT := PT - 1;
END_FOR;
FINDB_NUM := 0;

(* revision history
hm	6. oct 2006		rev 1.0
	original version

hm	29. feb 2008	rev 1.1
	improved performance

hm	29. mar. 2008	rev 1.2
	changed STRING to STRING(STRING_LENGTH)
*)
END_FUNCTION

(* POU String/FIND_CHAR, ST *)
FUNCTION FIND_CHAR : INT
VAR_INPUT
	str : STRING(STRING_LENGTH);
	pos : INT;
END_VAR
VAR
	i: INT;
	pt : POINTER TO ARRAY[1..255] OF BYTE;
	stop: INT;
	X: BYTE;
END_VAR

(*
version 1.3	21. oct. 2008
programmer 	hugo
tested by	tobias

find_char searches str and returns the starting position of the first character that is not a control character.
control characters are the ascii character 00 .. 31 and 127

*)
pt := ADR(str);
stop := LEN(str);
FOR i := MAX(pos,1) TO stop DO;
	X := pt^[i];
	IF X > 31 AND ((setup.EXTENDED_ASCII AND X <> 127) OR (NOT setup.EXTENDED_ASCII AND X < 127)) THEN
		FIND_CHAR := i;
		RETURN;
	END_IF;
END_FOR;
FIND_CHAR := 0;


(* revision history
hm	29. feb 2008	rev 1.0
	original version

hm	26. mar. 2008	rev 1.1
	char will now accept extended ascii

hm	29. mar. 2008	rev 1.2
	changed STRING to STRING(STRING_LENGTH)

hm	21. oct. 2008	rev 1.3
	changes setup constants
	optimized code
*)
END_FUNCTION

(* POU String/FIND_CTRL, ST *)
FUNCTION FIND_CTRL : INT
VAR_INPUT
	str : STRING(STRING_LENGTH);
	pos : INT;
END_VAR
VAR
	i: INT;
	pt : POINTER TO ARRAY[1..255] OF BYTE;
	stop: INT;
	x: BYTE;
END_VAR

(*
version 1.2	29. mar. 2008
programmer 	hugo
tested by		tobias

find_ctrl searches str and returns the starting position of a control character
control characters are the ascii character 00 .. 31 and 127.

*)
pt := ADR(str);
stop := LEN(str);
FOR i := MAX(pos,1) TO stop DO;
	x := PT^[I];
	IF x < 32 OR X = 127 THEN
		FIND_CTRL := i;
		RETURN;
	END_IF;
END_FOR;
FIND_CTRL := 0;


(* revision history
hm	29. feb 2008	rev 1.0
	original version

hm	26. mar. 2008	rev 1.1
	character 127 is now recognized as control

hm	29. mar. 2008	rev 1.2
	changed STRING to STRING(STRING_LENGTH)
*)
END_FUNCTION

(* POU String/FIND_NONUM, ST *)
FUNCTION FIND_NONUM : INT
VAR_INPUT
	str : STRING(STRING_LENGTH);
	pos : INT;
END_VAR
VAR
	i: INT;
	pt : POINTER TO ARRAY[1..255] OF BYTE;
	end: INT;
	X: BYTE;
END_VAR

(*
version 1.3	21. oct. 2008
programmer 	hugo
tested by	tobias

find_noNum searches str and returns the first position which is not a number.
a number is characterized by a letter "0..9" or "."

*)
pt := ADR(str);
end := LEN(str);
FOR i := MAX(pos,1) TO end DO;
	X := pt^[i];
	IF (X < 48 AND X <> 46) OR X > 57 THEN
		FIND_NONUM := i;
		RETURN;
	END_IF;
END_FOR;
FIND_NONUM := 0;


(* revision history
hm	6. oct. 2006	rev 1.0
	original version

hm	29. feb 2008	rev 1.1
	added input pos to start search at position

hm	29. mar. 2008	rev 1.2
	changed STRING to STRING(STRING_LENGTH)

hm	21. oct. 2008	rev 1.3
	optimized code

*)
END_FUNCTION

(* POU String/FIND_NUM, ST *)
FUNCTION FIND_NUM : INT
VAR_INPUT
	str : STRING(STRING_LENGTH);
	pos : INT;
END_VAR
VAR
	i : INT;
	pt : POINTER TO ARRAY[1..255] OF BYTE;
	stop : INT;
	X: BYTE;
END_VAR

(*
version 1.2	29. mar. 2008
programmer 	hugo
tested by		tobias

find_Num searches str and returns the starting position of a number
a number is characterized by a letter "0..9" or "."

*)
pt := ADR(str);
stop := LEN(str);
FOR i := MAX(pos,1) TO stop DO;
	X := pt^[i];
	IF (X > 47 AND X < 58) OR X = 46 THEN
		FIND_NUM := i;
		RETURN;
	END_IF;
END_FOR;
FIND_NUM := 0;


(* revision history
hm	6. oct. 2006	rev 1.0
	original version

hm	29. feb 2008	rev 1.1
	added input pos to start search at position

hm	29. mar. 2008	rev 1.2
	changed STRING to STRING(STRING_LENGTH)

*)
END_FUNCTION

(* POU String/FINDB, ST *)
FUNCTION FINDB : INT
VAR_INPUT
	str1 : STRING(STRING_LENGTH);
	str2 : STRING(STRING_LENGTH);
END_VAR
VAR
	pos: INT;
	length: INT;
END_VAR

(*
version 1.3	29. mar. 2008
programmer 	hugo
tested by		tobias

the function find searches an str1 for the presence of str2 and returns the first position of str1 of the last presence in instring.
the function is similar to find except it searches from the right to left.
 a 0 is returned if the string is not found.

*)
length := LEN(str2);
FOR pos := LEN(str1) - length + 1 TO 1 BY -1 DO
	IF MID(str1,length,pos) = str2 THEN
		FindB := pos;
		RETURN;
	END_IF;
END_FOR;
FindB := 0;

(* revision history
hm	6. oct 2006		rev 1.0
	original version

hm	15 dec 2007		rev 1.1
	changed code for better performance

hm	29. feb 2008	rev 1.2
	added findb := 0 for compatibility reasons

hm	29. mar. 2008	rev 1.3
	changed STRING to STRING(STRING_LENGTH)
*)
END_FUNCTION

(* POU String/FINDP, ST *)
FUNCTION FINDP : INT
VAR_INPUT
	str : STRING(STRING_LENGTH);
	src : STRING(STRING_LENGTH);
	pos: INT;
END_VAR
VAR
	i: INT;
	ls: INT;
	lx: INT;
	stp: INT;
END_VAR

(*
version 1.2	29. mar. 2008
programmer 	hugo
tested by	tobias

the function findP searches a string str for the occurence of src beginning at the position pos.

*)
ls := LEN(str);
lx := LEN(src);
IF ls < lx OR lx = 0 THEN RETURN; END_IF;
stp := ls - lx + 1;
FOR i := MAX(pos,1) TO stp DO
	IF MID(str,lx,i) = src THEN
		FINDP := i;
		RETURN;
	END_IF;
END_FOR;
FINDP := 0;

(* revision histroy
hm	4. feb. 2008	rev 1.0
	original release

hm	29. feb 2008	rev 1.1
	ADDED MAX(pos,1) in loop initialization

hm	29. mar. 2008	rev 1.2
	changed STRING to STRING(STRING_LENGTH)
*)	
END_FUNCTION

(* POU String/FLOAT_TO_REAL, ST *)
FUNCTION FLOAT_TO_REAL : REAL
VAR_INPUT
	FLT : STRING(20);
END_VAR
VAR
	pt : POINTER TO ARRAY[1..20] OF BYTE;
	i: INT;
	X: BYTE;
	sign: INT := 1;
	stop: INT;
	tmp: DINT;
	d : INT;
END_VAR

(*
version 1.3	23. oct. 2008
programmer 	hugo
tested by	oscat

FLOAT_TO_REAL converts a string to a REAL.
the function ignores all wrong characters.
the comma can be , or .
the exponent has to start with capital E or lowercase e .


*)
pt := ADR(FLT);
stop := LEN(FLT);

(* we first check for sign and exit if first number or dot is reached *)
FOR i := 1 TO stop DO
	X := pt^[i];
	IF X > 47 AND X < 58 OR X = 46 THEN
		EXIT;
	ELSIF X = 45 THEN
		(* code 45 is sign *)
		sign := -1;
	END_IF;
END_FOR;

(* now we scan numbers till end or dot or E is reached *)
FOR i := i TO stop DO
	X := pt^[i];
	IF X = 44 OR X = 46 OR X = 69 OR X = 101 THEN
		EXIT;
	(* calculate the value of the digit *)
	ELSIF X > 47 AND x < 58 THEN
		tmp := tmp * 10 + X - 48;
	END_IF;
END_FOR;

(* process the portion after the comma if comma or dot is reached exit if exponent starts *)
IF x = 44 OR X = 46 THEN
	FOR i := i + 1 TO stop DO
		X := pt^[i];
		IF X = 69 OR X = 101 THEN
			EXIT;
		ELSIF x > 47 AND x < 58 THEN
			tmp := tmp * 10 + X - 48;
			d := d - 1;
		END_IF;
	END_FOR;
END_IF;

(* process exponent if present *)
IF X = 69 OR X = 101 THEN
	d := d + DEC_TO_INT(RIGHT(FLT, stop - i));
END_IF;

FLOAT_TO_REAL :=  EXPN(10, d) * DINT_TO_REAL(TMP * SIGN);




(* revision histroy
hm	22. jun. 2008	rev 1.0
	original release

hm	2. oct. 2008	rev 1.1
	fixed an error, characters 8 and 9 would not be converted

hm	22. oct. 2008	rev 1.2
	last fix was not done correctly

hm	23. oct. 2008	rev 1.3
	optimzed code
*)	
END_FUNCTION

(* POU String/FSTRING_TO_BYTE, ST *)
FUNCTION FSTRING_TO_BYTE : BYTE
VAR_INPUT
	IN : STRING(12);
END_VAR


(*
version 1.1	20. sep. 2008
programmer 	hugo
tested by		oscat

FSTRING_TO_BYTE converts a formatted string into a byte.
the string can be of the form 2#01010, 8#7234, 16#2AD3 and 1234

*)
IF LEFT(IN, 2) = '2#' THEN
	(* we need to convert binary *)
	FSTRING_TO_BYTE := BIN_TO_BYTE(RIGHT(in, LEN(in) - 2));
ELSIF LEFT(in, 2) = '8#' THEN
	(* weneed to convert octals *)
	FSTRING_TO_BYTE := OCT_TO_BYTE(RIGHT(in, LEN(in) - 2));
ELSIF LEFT(in, 3) = '16#' THEN
	(* we need to convert hexadecimal *)
	FSTRING_TO_BYTE := HEX_TO_BYTE(RIGHT(in, LEN(in) - 3));
ELSE
	(* we assume decimal representation *)
	FSTRING_TO_BYTE := DEC_TO_BYTE(CLEAN(in,'0123456789'));
END_IF;


(* revision histroy
hm	18. jun. 2008	rev 1.0
	original release

hm	20. sep. 2008	rev 1.1
	changed length of input string from 20 to 12
*)	
END_FUNCTION

(* POU String/OCT_TO_BYTE, ST *)
FUNCTION OCT_TO_BYTE : BYTE
VAR_INPUT
	OCT : STRING(10);
END_VAR
VAR
	pt : POINTER TO BYTE;
	i: INT;
	X: BYTE;
	stop: INT;
END_VAR

(*
version 1.1	20. sep. 2008
programmer 	hugo
tested by		oscat

OCT_TO_BYTE converts a octagonal string into a byte.

*)
pt := ADR(oct);
stop := LEN(oct);
FOR I := 1 TO stop DO
	(* read the first character and subtract 48 to get value in decimal 0 = 48 *)
	x := pt^;
	(* calculate the value of the digit *)
	IF X > 47 AND x < 56 THEN
		OCT_TO_BYTE := SHL(OCT_TO_BYTE,3) + X - 48;
	END_IF;
	pt := pt + 1;
END_FOR;



(* revision histroy
hm	18. jun. 2008	rev 1.0
	original release

hm	20. sep. 2008	rev 1.1
	changed length of input string from 20 to 10

*)	
END_FUNCTION

(* POU String/HEX_TO_BYTE, ST *)
FUNCTION HEX_TO_BYTE : BYTE
VAR_INPUT
	HEX : STRING(5);
END_VAR
VAR
	pt : POINTER TO BYTE;
	i: INT;
	X: BYTE;
	stop: INT;
END_VAR

(*
version 1.1	20. sep. 2008
programmer 	hugo
tested by		oscat

HEX_TO_BYTE converts a Hexadecimal string into a byte.

*)
pt := ADR(hex);
stop := LEN(hex);
FOR I := 1 TO stop DO
	(* read the first character and subtract 48 to get value in decimal 0 = 48 *)
	x := pt^;
	(* calculate the value of the digit *)
	IF X > 47 AND x < 58 THEN
		HEX_TO_BYTE := SHL(HEX_TO_BYTE,4) + X - 48;
	ELSIF X > 64 AND X < 71 THEN
		HEX_TO_BYTE := SHL(HEX_TO_BYTE,4) + X - 55;
	ELSIF X > 96 AND X < 103 THEN
		HEX_TO_BYTE := SHL(HEX_TO_BYTE,4) + X - 87;
	END_IF;
	pt := pt + 1;
END_FOR;




(* revision histroy
hm	18. jun. 2008	rev 1.0
	original release

hm	20. sep.2008	rev 1.1
	changed length of input string from 20 to 5

*)	
END_FUNCTION

(* POU String/FSTRING_TO_DT, ST *)
FUNCTION FSTRING_TO_DT : DT
VAR_INPUT
	SDT : STRING(60);
	FMT : STRING(60);
END_VAR
VAR CONSTANT
	ignore: STRING(1) := '*';  (* ignore character is * *)
	fchar : STRING(1) := '#';  (* format character is # *)
END_VAR
VAR
	c: STRING(1);
	tmp: STRING(20);
	end: INT;
	dy : INT := 1970;
	dm : INT := 1;
	dd : INT := 1;
	th : INT;
	tm : INT;
	ts : INT;
END_VAR


(*
version 1.0	24. sep. 2008
programmer 	hugo
tested by	oscat

FSTRING_TO_DT converts Formatted String into a DT value.

*)
(* scan input string *)
WHILE fmt <> '' DO
	c := LEFT(fmt,1);
	IF c = ignore THEN
		(* skip ignore characters *)
		fmt := DELETE(fmt,1,1);
		sdt := DELETE(sdt,1,1);
	ELSIF C = fchar THEN
		(* format chracter found skip format char and read identifier *)
		(* store format identifier in c and skip to next char in fmt *)
		c := MID(fmt,1,2);
		fmt := DELETE(fmt,2,1);
		(* extract the substring until the end of sdt or to next char of fmt *)
		IF fmt = '' THEN
			tmp := sdt;
		ELSE
			(* serach for end of substring *)
			end := FIND(sdt, LEFT(fmt,1))-1;
			tmp := LEFT(sdt, end);
			sdt := DELETE(sdt, end,1);
		END_IF;
		(* extract information from substring *)
		IF c = 'Y' THEN
			dy := STRING_TO_INT(tmp);
			IF dy < 100 THEN dy := dy + 2000; END_IF;
		ELSIF c = 'M' THEN
			dm := STRING_TO_INT(tmp);
		ELSIF c = 'N' THEN
			dm := FSTRING_TO_MONTH(tmp,0);
		ELSIF c = 'D' THEN
			dd := STRING_TO_INT(tmp);
		ELSIF c = 'h' THEN
			th := STRING_TO_INT(tmp);
		ELSIF c = 'm' THEN
			tm := STRING_TO_INT(tmp);
		ELSIF c = 's' THEN
			ts := STRING_TO_INT(tmp);
		END_IF;
	ELSIF c = LEFT(sdt,1) THEN
		(* skip matching characters *)
		fmt := DELETE(fmt,1,1);
		sdt := DELETE(sdt,1,1);
	ELSE
		RETURN;
	END_IF;
END_WHILE;

FSTRING_TO_DT := SET_DT(dy,dm,dd,th,tm,ts);


(* revision histroy
hm	24. sep. 2008	rev 1.0
	original release


*)	
END_FUNCTION

(* POU String/FSTRING_TO_MONTH, ST *)
FUNCTION FSTRING_TO_MONTH : INT
VAR_INPUT
	MTH : STRING(20);
	LANG : INT;
END_VAR
VAR
	lx: INT;
END_VAR


(*
version 1.2	25. oct 2008
programmer 	hugo
tested by	oscat

FSTRING_TO_MONTH converts a string into a month, the string can be a name for the month or a number.
the function is language sensitve when LANG > 1 and checks for all languages when LANG = 0

*)
IF LANG = 0 THEN lx := LANGUAGE.DEFAULT; ELSE lx := MIN(LANG, LANGUAGE.LMAX); END_IF;
MTH := TRIM(mth);
MTH := CAPITALIZE(LOWERCASE(MTH));

FOR FSTRING_TO_MONTH := 1 TO 12 DO
	IF MTH = language.MONTHS[lx, FSTRING_TO_MONTH] THEN RETURN; END_IF;
	IF MTH = language.MONTHS3[lx, FSTRING_TO_MONTH] THEN RETURN; END_IF;
END_FOR;

(* since no name matched try to decode as integer *)
FSTRING_TO_MONTH := STRING_TO_INT(MTH);




(* revision histroy
hm	25. sep. 2008	rev 1.0
	original release

hm	19. oct. 2008	rev 1.1
	changed language setup constants

hm	25. oct. 2008	rev 1.2
	optimized code
*)	
END_FUNCTION

(* POU String/LOWERCASE, ST *)
FUNCTION LOWERCASE : STRING(STRING_LENGTH)
VAR_INPUT
	str : STRING(STRING_LENGTH);
END_VAR
VAR
	PT : POINTER TO BYTE;
	pos: INT;
	l: INT;
END_VAR

(*
version 1.3	29. mar. 2008
programmer 	hugo
tested by		tobias

lowercase returns str while all letters A..Z and Ä.Ö,Ü are converted to lowercase.

*)
PT := ADR(LOWERCASE);
lowercase := str;
l := LEN(str);
FOR pos := 1 TO l DO
	pt^ := TO_LOWER(pt^);
	PT := PT + 1;
END_FOR;

(* revision histroy
hm	6. oct. 2006	rev 1.0
	original release

hm	4. feb. 2008	rev 1.1
	improved performance
	added Ä.Ö,Ü

hm	6. mar. 2008	rev 1.2
	added support for exteded Ascii

hm	29. mar. 2008	rev 1.3
	changed STRING to STRING(STRING_LENGTH)
*)	
END_FUNCTION

(* POU String/TO_LOWER, ST *)
FUNCTION TO_LOWER : BYTE
VAR_INPUT
	IN : BYTE;
END_VAR


(*
version 1.2	25. oct 2008
programmer 	hugo
tested by		tobias

to_lower converts a character from uppercase to lowercase

*)
IF in > 64 AND in < 91 THEN
   TO_LOWER := in OR 16#20;
ELSIF (in > 191 AND in < 223) AND in <> 215 AND setup.EXTENDED_ASCII THEN
   TO_LOWER := in OR 16#20;
ELSE
   TO_LOWER := in;
END_IF;


(* revision history
hm	6. mar. 2008	rev 1.0
	original version

hm	19. oct. 2008	rev 1.1
	changed setup constants

ks	25. oct. 2008	rev 1.2
	optimized code
*)
END_FUNCTION

(* POU Time&Date/SET_DT, ST *)
FUNCTION SET_DT : DT
VAR_INPUT
	year : INT;
	month : INT;
	day : INT;
	hour : INT;
	minute : INT;
	second : INT;
END_VAR


(*
version 1.5	16 mar 2008
programmer 	hugo
tested by	tobias


creates a date output from year, month and day of month
year must be in the form of 4 digits ie 2006 or 1977.
*)
SET_DT := DWORD_TO_DT(DATE_TO_DWORD(SET_DATE(YEAR, MONTH, day)) + INT_TO_DWORD(SECOND) + INT_TO_DWORD(MINUTE) * 60 + INT_TO_DWORD(HOUR) * 3600);


(* revision history
hm	4. aug. 2006		rev 1.0
	original version

hm		19 sep. 2007	rev 1.1
	use function leap_year to calculate leap year, more exceptions are handled

hm		1. okt 2007		rev 1.2
	added step7 compatibility
	call function set_date

hm		8. oct 2007		rev 1.3
	deleted unused variables count and leap

hm		1. 11 2007		rev 1.4
	converted hour type integer to dword in calculation to avoid overrun on möller ecp4

hm		16. mar 2008	rev 1.5
	added type conversions to avoid warnings under codesys 3.0
*)
END_FUNCTION

(* POU Time&Date/SET_DATE, ST *)
FUNCTION SET_DATE : DATE
VAR_INPUT
	YEAR : INT;
	MONTH : INT;
	DAY : INT;
END_VAR
VAR
	count : INT;
END_VAR

(*
version 2.3	29. dec. 2011
programmer 	hugo
tested by	tobias

creates a date output from year, month and day of month   

*)
IF month > 2 THEN
	count := (month - 1) * 30;
	IF month > 7 THEN count := count + SHR(month - 3,1); ELSE count := count + SHR(month - 4,1); END_IF;
	(* chech for leap year and add one day if true *)
	IF SHL(year,14) = 0 THEN count := count + 1; END_IF;
ELSE
	count := (month - 1) * 31;
END_IF;

SET_DATE := DWORD_TO_DATE((INT_TO_DWORD(count + day - 1) + SHR(INT_TO_DWORD(year) * 1461 - 2878169, 2)) * 86400);


(* revision history
hm	4. aug. 2006	rev 1.0
	original version

hm	19 sep. 2007	rev 1.1
	use function leap_year to calculate leap year, more exceptions are handled

hm	1. okt	2007	rev 1.2
	added compatibility to step7

hm	16.dec 2007		rev 1.3
	changed code to improove performance

hm	3. jan. 2008	rev 1.4
	further improvements in performance

hm	16. mar. 2008	rev 1.5
	added type conversions to avoid warnings under codesys 3.0

hm	7. apr. 2008	rev 1.6
	deleted unused step7 code

hm	14. oct. 2008	rev 1.7
	optimized code for better performance

hm	25. oct. 2008	rev 2.0
	new code using setup constants

hm	16. nov. 2008	rev 2.1
	added typecasts to avoid warnings

hm	22. jan. 2011	rev 2.2
	improved performance

hm	29. dec. 2011	rev 2.3
	improved performance
*)
END_FUNCTION

(* POU String/FSTRING_TO_DWORD, ST *)
FUNCTION FSTRING_TO_DWORD : DWORD
VAR_INPUT
	IN : STRING(40);
END_VAR


(*
version 1.1	20. sep. 2008
programmer 	hugo
tested by		oscat

FSTRING_TO_BYTE converts a formatted string into a byte.
the string can be of the form 2#01010, 8#7234, 16#2AD3 and 1234

*)
IF LEFT(IN, 2) = '2#' THEN
	(* we need to convert binary *)
	FSTRING_TO_DWORD := BIN_TO_DWORD(RIGHT(in, LEN(in) - 2));
ELSIF LEFT(in, 2) = '8#' THEN
	(* weneed to convert octals *)
	FSTRING_TO_DWORD := OCT_TO_DWORD(RIGHT(in, LEN(in) - 2));
ELSIF LEFT(in, 3) = '16#' THEN
	(* we need to convert hexadecimal *)
	FSTRING_TO_DWORD := HEX_TO_DWORD(RIGHT(in, LEN(in) - 3));
ELSE
	(* we assume decimal representation *)
	FSTRING_TO_DWORD := DEC_TO_DWORD(CLEAN(in,'0123456789'));
END_IF;


(* revision histroy
hm	18. jun. 2008	rev 1.0
	original release

hm	20. sep. 2008	rev 1.1
	changed length of input dtring from 20 to 40


*)	
END_FUNCTION

(* POU String/OCT_TO_DWORD, ST *)
FUNCTION OCT_TO_DWORD : DWORD
VAR_INPUT
	OCT : STRING(20);
END_VAR
VAR
	pt : POINTER TO BYTE;
	i: INT;
	X: BYTE;
	stop: INT;
END_VAR

(*
version 1.0	18. jun 2008
programmer 	hugo
tested by	oscat

OCT_TO_DWORD converts a octagonal string into a dword.

*)
pt := ADR(oct);
stop := LEN(oct);
FOR I := 1 TO stop DO
	(* read the first character and subtract 48 to get value in decimal 0 = 48 *)
	x := pt^;
	(* calculate the value of the digit *)
	IF X > 47 AND x < 56 THEN
		OCT_TO_DWORD := SHL(OCT_TO_DWORD,3) + X - 48;
	END_IF;
	pt := pt + 1;
END_FOR;




(* revision histroy
hm	18. jun. 2008	rev 1.0
	original release


*)	
END_FUNCTION

(* POU String/HEX_TO_DWORD, ST *)
FUNCTION HEX_TO_DWORD : DWORD
VAR_INPUT
	Hex : STRING(20);
END_VAR
VAR
	pt : POINTER TO BYTE;
	i: INT;
	X: BYTE;
	stop: INT;
END_VAR

(*
version 1.4	18. jun. 2008
programmer 	hugo
tested by	tobias

HEX_TO_DWORD converts a Hexadecimal string into a DWORD.

*)
pt := ADR(hex);
stop := LEN(hex);
FOR I := 1 TO stop DO
	(* read the first character and subtract 48 to get value in decimal 0 = 48 *)
	x := pt^;
	(* calculate the value of the digit *)
	IF X > 47 AND x < 58 THEN
		HEX_TO_DWORD := SHL(HEX_TO_DWORD,4) + X - 48;
	ELSIF X > 64 AND X < 71 THEN
		HEX_TO_DWORD := SHL(HEX_TO_DWORD,4) + X - 55;
	ELSIF X > 96 AND X < 103 THEN
		HEX_TO_DWORD := SHL(HEX_TO_DWORD,4) + X - 87;
	END_IF;
	pt := pt + 1;
END_FOR;



(* revision histroy
hm	2.10.2007		rev 1.0
	original release

hm	19.11.2007		rev 1.1
	changed type of function from int to dword

hm 	4. mar 2008		rev 1.2
	added support for a..f and return 0 for invalid string

hm	29. mar. 2008	rev 1.3
	changed STRING to STRING(8)

hm	18. jun. 2008	rev 1.4
	changed input hex to STRING(20)
	function now ignores wrong characters
*)	
END_FUNCTION

(* POU String/FSTRING_TO_WEEK, ST *)
FUNCTION FSTRING_TO_WEEK : BYTE
VAR_INPUT
	WEEK : STRING(60);
	LANG : INT;
END_VAR
VAR
	pos: INT;
END_VAR


(*
version 1.1	25. oct. 2008
programmer 	hugo
tested by	oscat

FSTRING_TO_WEEK converts a list of weekdays into a byte where each bit represents a day of the week.
bit 6 = mo, 0 = su;

*)
pos := FIND(WEEK, ',');
WHILE pos > 0 DO
	FSTRING_TO_WEEK := FSTRING_TO_WEEK OR SHR(BYTE#128, FSTRING_TO_WEEKDAY(MID(WEEK, pos - 1, 1), LANG));
	WEEK := RIGHT(WEEK, LEN(Week) - pos);
	pos := FIND(WEEK, ',');
END_WHILE;
FSTRING_TO_WEEK := (FSTRING_TO_WEEK OR SHR(BYTE#128, FSTRING_TO_WEEKDAY(WEEK, LANG))) AND BYTE#127;


(* revision histroy
hm	18. jun. 2008	rev 1.0
	original release

hm	25. oct. 2008	rev 1.1
	using language defauls and input lang
*)	
END_FUNCTION

(* POU String/FSTRING_TO_WEEKDAY, ST *)
FUNCTION FSTRING_TO_WEEKDAY : INT
VAR_INPUT
	WDAY : STRING(20);
	LANG : INT;
END_VAR
VAR
	tmp: STRING(2);
	i: INT;
	ly: INT;
END_VAR


(*
version 1.2	25. oct. 2008
programmer 	hugo
tested by	oscat

FSTRING_TO_WEEKDAY converts a weekday string into an integer 1..7.

*)
IF LANG = 0 THEN ly := LANGUAGE.DEFAULT; ELSE ly := MIN(LANG, LANGUAGE.LMAX); END_IF;
(* tmp needs to be calculated first otherwise find can return wrong values *)
tmp := TRIM(wday);
tmp := CAPITALIZE(LOWERCASE(tmp));
FOR i := 1 TO 7 DO
	IF language.WEEKDAYS2[ly, i] = tmp THEN
		FSTRING_TO_WEEKDAY := i;
		RETURN;
	END_IF;
END_FOR;
FSTRING_TO_WEEKDAY := STRING_TO_INT(WDAY);




(* revision histroy
hm	18. jun. 2008	rev 1.0
	original release

hm	18. jul. 2008	rev 1.1
	changed nested call of left(trim()) for compatibility reasons

hm	25. oct. 2008	rev 1.2
	using language constants
*)	
END_FUNCTION

(* POU String/IS_ALNUM, ST *)
FUNCTION IS_ALNUM : BOOL
VAR_INPUT
	str : STRING(STRING_LENGTH);
END_VAR
VAR
	L: INT;
	pt : POINTER TO BYTE;
	pos: INT;
END_VAR

(*
version 1.1	29. mar. 2008
programmer 		kurt
tested by		hugo

ISC_ALNUM testet ob in einem string nur Zahlen 0..9 vorkommen.

*)
PT := ADR(str);
L := LEN(str);
FOR pos := 1 TO L DO
	IF NOT (ISC_ALPHA(pt^) OR ISC_NUM(pt^)) THEN
		IS_ALNUM := FALSE;
		RETURN;
	END_IF;
    	PT := PT + 1;
END_FOR;
IS_ALNUM := L > 0;


(* revision history
hm	29. feb 2008	rev 1.0
	original version

hm	29. mar. 2008	rev 1.1
	changed STRING to STRING(STRING_LENGTH)
*)
END_FUNCTION

(* POU String/ISC_ALPHA, ST *)
FUNCTION ISC_ALPHA : BOOL
VAR_INPUT
	IN : BYTE;
END_VAR


(*
version 1.1	19. oct. 2008
programmer 	oscat
tested by	oscat

ISC_ALPHA checks if a character is a..z or A..Z.

*)
IF setup.EXTENDED_ASCII THEN
	ISC_ALPHA := (in > 64 AND in < 91) OR (in > 191  AND in <> 215 AND in <> 247) OR (in > 96 AND in < 123);
ELSE
	ISC_ALPHA := (IN > 64 AND IN < 91) OR (in > 96 AND in < 123);
END_IF;

(* revision history
hm	6. mar. 2008	rev 1.0
	original version

hm	19. oct. 2008	rev 1.1
	changes setup constants
*)
END_FUNCTION

(* POU String/ISC_NUM, ST *)
FUNCTION ISC_NUM : BOOL
VAR_INPUT
	IN : BYTE;
END_VAR


(*
version 1.0	6. mar 2008
programmer 	oscat
tested by		hugo

ISC_NUM checks if a character is 0..9.

*)
ISC_NUM := IN > 47 AND IN < 58;

(* revision history
hm		6. mar. 2008	rev 1.0
	original version

*)
END_FUNCTION

(* POU String/IS_ALPHA, ST *)
FUNCTION IS_ALPHA : BOOL
VAR_INPUT
	str : STRING(STRING_LENGTH);
END_VAR
VAR
	L: INT;
	pt : POINTER TO BYTE;
	pos: INT;
END_VAR

(*
version 1.1	29. mar. 2008
programmer 		kurt
tested by		hugo

IS_ALPHA testet ob in einem string nur Zeichen a-z oder A - Z vorkommen.

*)
PT := ADR(str);
L := LEN(str);
FOR pos := 1 TO L DO
	IF NOT ISC_ALPHA(pt^) THEN
		IS_ALPHA := FALSE;
		RETURN;
	END_IF;
    	PT := PT + 1;
END_FOR;
IS_ALPHA := L > 0;


(* revision history
hm	29. feb 2008	rev 1.0
	original version

hm	29. mar. 2008	rev 1.1
	changed STRING to STRING(STRING_LENGTH)
*)
END_FUNCTION

(* POU String/IS_CC, ST *)
FUNCTION IS_CC : BOOL
VAR_INPUT
	str : STRING(STRING_LENGTH);
	cmp : STRING(STRING_LENGTH);
END_VAR
VAR
	L: INT;
	pos: INT;
END_VAR

(*
version 1.1	29. mar. 2008
programmer 	Tobias
tested by	hugo

ISC_CC testet ob ein string nur aus Zeichen des Strings CMP besteht.

*)
L := LEN(str);
FOR pos := 1 TO L DO
	IF FIND(CMP,MID(str,1,pos)) = 0 THEN RETURN; END_IF;
END_FOR;
IS_CC := L > 0;



(* revision history
hm	19. mar 2008	rev 1.0
	original version

hm	29. mar. 2008	rev 1.1
	changed STRING to STRING(STRING_LENGTH)
*)
END_FUNCTION

(* POU String/IS_CTRL, ST *)
FUNCTION IS_CTRL : BOOL
VAR_INPUT
	STR : STRING(STRING_LENGTH);
END_VAR
VAR
	L: INT;
	pt : POINTER TO BYTE;
	pos: INT;
END_VAR

(*
version 1.1	29. mar 2008
programmer 		kurt
tested by		hugo

IS_CTRL testet ob in einem string nur Steuerzeichen (Char < 32) vorkommen.

*)
PT := ADR(str);
L := LEN(str);
FOR pos := 1 TO L DO
	IF NOT (ISC_CTRL(pt^)) THEN
		IS_CTRL := FALSE;
		RETURN;
	END_IF;
    	PT := PT + 1;
END_FOR;
IS_CTRL := L > 0;


(* revision history
hm	29. feb. 2008	rev 1.0
	original version

hm	29. mar. 2008	rev 1.1
	changed STRING to STRING(STRING_LENGTH)
*)
END_FUNCTION

(* POU String/ISC_CTRL, ST *)
FUNCTION ISC_CTRL : BOOL
VAR_INPUT
	IN : BYTE;
END_VAR


(*
version 1.0	6. mar 2008
programmer 	oscat
tested by		hugo

ISC_ALPHA checks if a character is a control character.

*)
ISC_CTRL := IN < 32 OR IN = 127;

(* revision history
hm		6. mar. 2008	rev 1.0
	original version

*)
END_FUNCTION

(* POU String/IS_HEX, ST *)
FUNCTION IS_HEX : BOOL
VAR_INPUT
	str : STRING(STRING_LENGTH);
END_VAR
VAR
	L: INT;
	pt : POINTER TO BYTE;
	pos: INT;
END_VAR

(*
version 1.1	29. mar. 2008
programmer 		kurt
tested by		hugo

IS_HEX testet ob in einem string nur Zahlen 0..9 oder A..F oder a..f  vorkommen.

*)
PT := ADR(str);
L := LEN(str);
FOR pos := 1 TO L DO
	IF NOT (ISC_HEX(pt^)) THEN
		IS_HEX := FALSE;
		RETURN;
	END_IF;
    	PT := PT + 1;
END_FOR;
IS_HEX := L > 0;


(* revision history
hm	29. feb 2008	rev 1.0
	original version

hm	29. mar. 2008	rev 1.1
	changed STRING to STRING(STRING_LENGTH)
*)
END_FUNCTION

(* POU String/ISC_HEX, ST *)
FUNCTION ISC_HEX : BOOL
VAR_INPUT
	IN : BYTE;
END_VAR


(*
version 1.0	6. mar 2008
programmer 	oscat
tested by		hugo

ISC_HEX checks if a character is 0..9, A..F, a..f.

*)
ISC_HEX := (IN > 47 AND IN < 58) OR (IN > 64 AND IN < 71) OR (IN > 96 AND IN < 103);

(* revision history
hm		6. mar. 2008	rev 1.0
	original version

*)
END_FUNCTION

(* POU String/IS_LOWER, ST *)
FUNCTION IS_LOWER : BOOL
VAR_INPUT
	str : STRING(STRING_LENGTH);
END_VAR
VAR
	l: INT;
	pt : POINTER TO BYTE;
	pos: INT;
END_VAR

(*
version 1.1	29. mar. 2008
programmer 		kurt
tested by		hugo

IS_LOWER testet ob in einem string nur kleinbuchstaben vorkommen.

*)
PT := ADR(str);
L := LEN(str);
FOR pos := 1 TO L DO
	IF NOT (ISC_LOWER(pt^)) THEN
		IS_LOWER := FALSE;
		RETURN;
	END_IF;
    	PT := PT + 1;
END_FOR;
IS_LOWER := L > 0;


(* revision history
hm	29. feb 2008	rev 1.0
	original version

hm	29. mar. 2008	rev 1.1
	changed STRING to STRING(STRING_LENGTH)
*)
END_FUNCTION

(* POU String/ISC_LOWER, ST *)
FUNCTION ISC_LOWER : BOOL
VAR_INPUT
	IN : BYTE;
END_VAR


(*
version 1.1	19. oct. 2008
programmer 	hugo
tested by	oscat

isc_lower checks if a character is lowercase.

*)
IF setup.EXTENDED_ASCII THEN
	ISC_LOWER := ((in > 96) AND (in < 123)) OR ((in > 222) AND (in <> 247));
ELSE
	ISC_LOWER := ((in > 96) AND (in < 123));
END_IF;

(* revision history
hm	6. mar. 2008	rev 1.0
	original version

hm	19. oct. 2008	rev 1.1
	changes setup constants
*)
END_FUNCTION

(* POU String/IS_NCC, ST *)
FUNCTION IS_NCC : BOOL
VAR_INPUT
	str : STRING(STRING_LENGTH);
	cmp : STRING(STRING_LENGTH);
END_VAR
VAR
	L: INT;
	pos: INT;
END_VAR

(*
version 1.1	29. mar. 2008
programmer 	Tobias
tested by		hugo

IS_NCC testet ob in einem string keine Zeichen des Strings CMP enthalten sind.

*)
L := LEN(str);
FOR pos := 1 TO L DO
	IF FIND(CMP,MID(str,1,pos)) > 0 THEN RETURN; END_IF;
END_FOR;
IS_NCC := TRUE;



(* revision history
hm	19. mar 2008	rev 1.0
	original version

hm	29. mar. 2008	rev 1.1
	changed STRING to STRING(STRING_LENGTH)
*)
END_FUNCTION

(* POU String/IS_NUM, ST *)
FUNCTION IS_NUM : BOOL
VAR_INPUT
	str : STRING(STRING_LENGTH);
END_VAR
VAR
	L : INT;
	pt : POINTER TO BYTE;
	pos: INT;
END_VAR

(*
version 1.1	29. mar. 2008
programmer 		kurt
tested by		hugo

IS_NUM testet ob in einem string nur Zahlen 0..9 vorkommen.

*)
PT := ADR(str);
L := LEN(str);
FOR pos := 1 TO L DO
	IF NOT (ISC_NUM(pt^)) THEN
		IS_NUM := FALSE;
		RETURN;
	END_IF;
    	PT := PT + 1;
END_FOR;
IS_NUM := L > 0;


(* revision history
hm	29. feb 2008	rev 1.0
	original version

hm	29. mar. 2008	rev 1.1
	changed STRING to STRING(STRING_LENGTH)
*)
END_FUNCTION

(* POU String/IS_UPPER, ST *)
FUNCTION IS_UPPER : BOOL
VAR_INPUT
	str : STRING(STRING_LENGTH);
END_VAR
VAR
	L: INT;
	pt : POINTER TO BYTE;
	pos: INT;
END_VAR

(*
version 1.1	29. mar. 2008
programmer 		kurt
tested by		hugo

IS_UPPER testet ob in einem string keine Kleinbuchstaben vorkommen.

*)
PT := ADR(str);
L := LEN(str);
FOR pos := 1 TO L DO
	IF NOT (ISC_UPPER(pt^)) THEN
		IS_UPPER := FALSE;
		RETURN;
	END_IF;
    	PT := PT + 1;
END_FOR;
IS_UPPER := L > 0;


(* revision history
hm	29. feb 2008	rev 1.0
	original version

hm	29. mar. 2008	rev 1.1
	changed STRING to STRING(STRING_LENGTH)
*)
END_FUNCTION

(* POU String/ISC_UPPER, ST *)
FUNCTION ISC_UPPER : BOOL
VAR_INPUT
	IN : BYTE;
END_VAR


(*
version 1.1	19. oct. 2008
programmer 	hugo
tested by	oscat

ISC_upper checks if a character is uppercase

*)
IF setup.EXTENDED_ASCII THEN
	ISC_UPPER :=  ((in > 64) AND (in < 91)) OR (((in > 191) AND (in < 223)) AND (in <> 215));
ELSE
	ISC_UPPER := ((in > 64) AND (in < 91));
END_IF;


(* revision history
hm	6. mar. 2008	rev 1.0
	original version

hm	19. oct. 2008	rev 1.1
	changes setup constants

*)
END_FUNCTION

(* POU String/MESSAGE_4R, ST *)
FUNCTION_BLOCK MESSAGE_4R
VAR_INPUT
	M0 : STRING(STRING_LENGTH);
	M1 : STRING(STRING_LENGTH);
	M2 : STRING(STRING_LENGTH);
	M3 : STRING(STRING_LENGTH);
	MM : INT := 3;
	ENQ : BOOL := TRUE;
	CLK : BOOL := TRUE;
	T1 : TIME := T#3s;
END_VAR
VAR_OUTPUT
	MX : STRING(STRING_LENGTH);
	MN : INT;
	TR : BOOL;
END_VAR
VAR
	timer : TON;
	edge: BOOL;
END_VAR

(*
version 1.1	27. oct. 2008
programmer 	hugo
tested by	tobias

this function generates a rotation meassage with up to 4 strings.
on each rising edge of EN the next message in line will be displayed.
when EN stays high longer then one cycle, the next message will be displayed automatically after the time T1 is elapsed.
the output MX is the generated message and CX is a counter 0..3 signaling the current message displayed.
the displayed messages are 0 .. MM.

*)
(* check for rising edge on EN *)
TR := FALSE;
IF ENQ THEN
	IF (NOT edge AND clk) OR timer.q THEN
			MN := INC1(MN, MM);
			TR := TRUE;
			timer(in := FALSE);
			CASE MN OF
				0 : MX := M0;
				1 : MX := M1;
				2 : MX := M2;
				3 : MX := M3;
			END_CASE;
	END_IF;
	edge := clk;
	timer( in := CLK, pt := T1);
ELSE
	MX := '';
	MN := 0;
END_IF;




(* revision history
hm	8. oct. 2008	rev 1.0
	original version

hm	27. oct. 2008	rev 1.1
	changed _INC to INC1

*)
END_FUNCTION_BLOCK

(* POU String/MESSAGE_8, ST *)
FUNCTION_BLOCK MESSAGE_8
VAR_INPUT
	IN1 : BOOL;
	IN2 : BOOL;
	IN3 : BOOL;
	IN4 : BOOL;
	IN5 : BOOL;
	IN6 : BOOL;
	IN7 : BOOL;
	IN8 : BOOL;
END_VAR
VAR_INPUT CONSTANT
	S1 : STRING(STRING_LENGTH);
	S2 : STRING(STRING_LENGTH);
	S3 : STRING(STRING_LENGTH);
	S4 : STRING(STRING_LENGTH);
	S5 : STRING(STRING_LENGTH);
	S6 : STRING(STRING_LENGTH);
	S7 : STRING(STRING_LENGTH);
	S8 : STRING(STRING_LENGTH);
END_VAR
VAR_OUTPUT
	M : STRING(STRING_LENGTH);
END_VAR


(*
version 1.1	29. mar. 2008
programmer 	hugo
tested by	tobias

this function generates one out of 4 messages specified by S1 .. S8.
the selected message will be presented at the output M.
In1 has higher priority then In2 which has higher priority then IN3 and in8 has the lowest priority.
*)
(* check if an alarm is present if yes set the output M otherwise clear M *)
IF in1 THEN
	M := S1;
ELSIF in2 THEN
	M := S2;
ELSIF in3 THEN
	M := S3;
ELSIF in4 THEN
	M := S4;
ELSIF in5 THEN
	M := S5;
ELSIF in6 THEN
	M := S6;
ELSIF in7 THEN
	M := S7;
ELSIF in8 THEN
	M := S8;
ELSE
	M := '';
END_IF;

(* revision history
hm	26.12.2007		rev 1.0
	original version

hm	29. mar. 2008	rev 1.1
	changed STRING to STRING(STRING_LENGTH)
*)
END_FUNCTION_BLOCK

(* POU String/MIRROR, ST *)
FUNCTION MIRROR : STRING(STRING_LENGTH)
VAR_INPUT
	str : STRING(STRING_LENGTH);
END_VAR
VAR
	pi : POINTER TO ARRAY[1..255] OF BYTE;
	po : POINTER TO BYTE;
	lx: INT;
	i: INT;
END_VAR

(*
version 1.1	29. mar. 2008
programmer 	hugo
tested by	tobias

this function reverses an input string.

*)
pi := ADR(str);
po := ADR(mirror);
lx := LEN(str);
FOR i := lx TO 1 BY - 1 DO
	po^ := pi^[i];
	po := po + 1;
END_FOR;
(* close output string *)
po^:= 0;


(* revision histroy
hm	4. feb. 2008	rev 1.0
	original release

hm	29. mar. 2008	rev 1.1
	changed STRING to STRING(STRING_LENGTH)
*)	
END_FUNCTION

(* POU String/REAL_TO_STRF, ST *)
FUNCTION REAL_TO_STRF : STRING(20)
VAR_INPUT
	IN : REAL;
	N : INT;
	D : STRING(1);
END_VAR
VAR
	O: REAL;
	i: INT;
END_VAR

(*
version 1.8	2. jan 2012
programmer 	hugo
tested by	oscat

Real_to_strf converts a Real to a fixed length String.
the string will be filles with zeroes to achieve the fixed length N after the decimal separator.
the input parameter specifies the decimal separator to be used in the output string.

*)
(* LIMIT N to 0 .. 7 *)
N := LIMIT(0,N,7);
(* round the input to N digits and convert to string *)
O := ABS(in) * EXP10(N);
REAL_TO_STRF := DINT_TO_STRING(REAL_TO_DINT(O));
(* add zeroes in front to make sure sting is at least 8 digits long *)
FOR i := LEN(REAL_TO_STRF) TO N DO REAL_TO_STRF := CONCAT('0', REAL_TO_STRF); END_FOR;
(* add a dot if n > 0 *)
IF n > 0 THEN REAL_TO_STRF := INSERT(REAL_TO_STRF, D, LEN(REAL_TO_STRF) - N); END_IF;
(* add a minus sign if in is negative *)
IF in < 0 THEN REAL_TO_STRF := CONCAT('-', REAL_TO_STRF); END_IF;


(* revision history
hm	26 jan 2007	rev 1.0
	original version

hm	20. nov. 2007	rev 1.1
	when N=0 ther will be no dot at the end of the string.

hm	15. dec. 2007	rev 1.2
	changed code for better performance

hm	4. mar. 2008	rev 1.3
	result is now rounded instead of trunc

hm	20. mar. 2008	rev 1.4
	changed trunc to real_to_dint because trunc was generating wrong values on wago 842

hm	29. mar. 2008	rev 1.5
	changed STRING to STRING(20)

hm	4. apr. 2008	rev 1.6
	added variable O to avoid an error uner CoDeSys SP PLCWinNT V2.4

hm	27. feb. 2009	rev 1.7
	added a missing zero for IN < 1

hm 2. jan 2012	rev 1.8
	added input parameter D to specify decimal separator
*)
END_FUNCTION

(* POU String/REPLACE_ALL, ST *)
FUNCTION REPLACE_ALL : STRING(STRING_LENGTH)
VAR_INPUT
	str : STRING(STRING_LENGTH);
	src : STRING(STRING_LENGTH);
	rep : STRING(STRING_LENGTH);
END_VAR
VAR
	pos: INT;
	lp : INT;
	lx : INT;
END_VAR

(*
version 1.1	29. mar. 2008
programmer 	hugo
tested by	tobias

the function replace_all replaces all occurences of src in str and replaces them by rep.

*)
REPLACE_ALL := str;
lx := LEN(src);
lp := LEN(rep);
pos := FINDP(REPLACE_ALL, src, 1);
WHILE pos > 0 DO
	REPLACE_ALL := REPLACE(REPLACE_ALL,rep,lx, pos);
	pos := FINDP(REPLACE_ALL, src, pos + lp);
END_WHILE;

(* revision histroy
hm	4. feb. 2008	rev 1.0
	original release

hm	29. mar. 2008	rev 1.1
	changed STRING to STRING(STRING_LENGTH)
*)	
END_FUNCTION

(* POU String/REPLACE_CHARS, ST *)
FUNCTION REPLACE_CHARS : STRING(STRING_LENGTH)
VAR_INPUT
	STR : STRING(STRING_LENGTH);
	SRC : STRING;
	REP : STRING;
END_VAR
VAR
	a, b : INT;
	c: STRING(1);
	stp: INT;
END_VAR

(*
version 1.0		14. may. 2008
programmer 		hugo
tested by			hugo

REPLACE_CHARS erstezt alle character die im string src aufgeführt sind mit dem an der selben stelle im string rep gelisteten character.

*)
REPLACE_CHARS := STR;
(* make sure rep and src are of same length and length is > 0 *)
a := LEN(src);
b := LEN(rep);
IF a < b THEN
	rep := LEFT(rep, a);
ELSIF b < a THEN
	src := LEFT(src, b);
END_IF;

(* search the string and replace if necessary *)
stp := LEN(str);
FOR a := 1 TO stp DO
	c := MID(REPLACE_CHARS, 1, a);
	b := FIND(src, c);
	IF b > 0 THEN
		REPLACE_CHARS := REPLACE(REPLACE_CHARS, MID(rep, 1, b), 1, a);
	END_IF;
END_FOR;



(* revision history
hm	14. may. 2008	rev 1.0
	original version

*)
END_FUNCTION

(* POU String/REPLACE_UML, ST *)
FUNCTION REPLACE_UML : STRING(STRING_LENGTH)
VAR_INPUT
	str : STRING(STRING_LENGTH);
END_VAR
VAR
	L : INT;
	pt : POINTER TO BYTE;
	pto : POINTER TO BYTE;
	ptm : POINTER TO BYTE;
	pt1, pt2 : POINTER TO BYTE;
	su : STRING(2);
	pos : INT;
END_VAR

(*
version 1.1	29. mar. 2008
programmer 		kurt
tested by		hugo

REPLACE_UML replaces all occurences of Ä,Ö,Ü and ä,ö,ü,ß with Ae, ae, Oe, oe, Ue, ue and ss.

*)
PT := ADR(str);
pto := ADR(REPLACE_UML);
ptm := pto + INT_TO_DWORD(string_length);
pt1 := ADR(su);
pt2 := pt1 + 1;
L := LEN(str);
WHILE pos < L AND pos < string_length DO
	IF pt^ < 127 THEN
		(* no uml character simlply copy the character*)
		pto^ := pt^;
	ELSE
		(* convert the uml character *)
		su := TO_UML(pt^);
		(* we must make sure pointer are not out of range *)
		pto^ := pt1^;
		IF pto < ptm AND pt2^ > 0 THEN
			pto := pto + 1;
			pto^ := pt2^;
		END_IF;
	END_IF;
	(* increment pointers *)
	pt := pt + 1;
	pto := pto + 1;
	pos := pos + 1;
END_WHILE;

(* properly close the output string *)
pto^ := 0;


(* revision history
hm	29. feb 2008	rev 1.0
	original version

hm	29. mar. 2008	rev 1.1
	changed STRING to STRING(STRING_LENGTH)
	new code to avoid pointer out of range
	use new function to_uml
*)
END_FUNCTION

(* POU String/TO_UML, ST *)
FUNCTION TO_UML : STRING(2)
VAR_INPUT
	IN : BYTE;
END_VAR


(*
version 1.1	17. dec. 2008
programmer 		hugo
tested by		tobias

to_uml converts a character above 127 to a two digit character below 127.
the character Ä is converted to Ae

*)
CASE in OF
	196:	(* Ä *)
		TO_UML := 'Ae';
	214:	(* Ö *)
		TO_UML := 'Oe';
	220:	(* Ü *)
		TO_UML := 'Ue';
	223:	(* ß *)
		TO_UML := 'ss';
	228:	(* ä *)
		TO_UML := 'ae';
	246:	(* ö *)
		TO_UML := 'oe';
	252:	(* ü *)
		TO_UML := 'ue';
ELSE
	TO_UML := CHR_TO_STRING(IN);
END_CASE;



(* revision history
hm	29. mar. 2008	rev 1.0
	original version

hm	17. dec. 2008	rev 1.1
	changes name of function chr to chr_to_string

*)
END_FUNCTION

(* POU String/TICKER, ST *)
FUNCTION_BLOCK TICKER

VAR_INPUT
	N : INT;
	PT : TIME;
END_VAR

VAR_IN_OUT
	Text : STRING(STRING_LENGTH);
END_VAR

VAR_OUTPUT
	Display : STRING(STRING_LENGTH);
END_VAR
VAR
	delay : TP;
	step : INT;
END_VAR

(*
version 1.2	29. mar. 2008
programmer 	hugo
tested by		tobias

Ticker sends a substring of text with length N every TD Milliseconds to generate a ticker. 

*)
(* generate next ticker when delay is low *)
IF N < LEN(text) THEN
	IF NOT delay.Q THEN
		(* increase step for next tick *)
		step := step + 1;
		IF step > LEN(text) THEN step := 1; END_IF;
		(* extract dispay from text *)
		display := MID(text, N, step);
		(* set delay timer for next tick *)
		delay(in := TRUE, PT := PT);
	ELSE;
		(* execute delay timer *)
		delay(in := FALSE);
	END_IF;
ELSE
	display := text;
END_IF;
(* revision history
hm	4. dec. 2007	rev 1.0
	original version

hm	15. dec. 2007	rev 1.1
	step now starts at 1 instaed of 0

hm	29. mar. 2008	rev 1.2
	changed STRING to STRING(STRING_LENGTH)
*)
END_FUNCTION_BLOCK

(* POU String/TRIM1, ST *)
FUNCTION TRIM1 : STRING(STRING_LENGTH)
VAR_INPUT
	str : STRING(STRING_LENGTH);
END_VAR
VAR
	pos: INT;
END_VAR

(*
version 1.2	29. mar. 2008
programmer 	hugo
tested by		tobias

the function replaces all multiple blanks within a string by only one blank.
leading and ending blanks will be deleted

*)
TRIM1 := str;
REPEAT
	pos := FIND(trim1,'  ');
	IF pos > 0 THEN TRIM1 := REPLACE(TRIM1,' ',2,pos); END_IF;
UNTIL pos = 0	END_REPEAT;
(* beginning and ending blanks need to be stripped off *)
IF LEFT(trim1,1) = ' ' THEN trim1 := DELETE(trim1,1,1); END_IF;
IF RIGHT(trim1,1) = ' ' THEN trim1 := DELETE(trim1,1,LEN(trim1)); END_IF;


(* revision histroy
hm	4. feb. 2008    rev 1.0
	original release

hm	20. mar. 2008	rev 1.1
	avoid to call replace with pos = 0 because some systems will produce an error

hm	29. mar. 2008	rev 1.2
	changed STRING to STRING(STRING_LENGTH)
*)
END_FUNCTION

(* POU String/TRIME, ST *)
FUNCTION TRIME : STRING(string_length)
VAR_INPUT
	str : STRING(STRING_LENGTH);
END_VAR


(*
version 1.0	28. mar. 2008
programmer 	hugo
tested by	tobias

this function deletes all leading and ending blanks of a string.

*)
TRIME := str;
(* beginning blanks need to be stripped off *)
WHILE LEFT(TRIME,1) = ' ' DO
	TRIME := DELETE(TRIME,1,1);
END_WHILE;

(* ending blanks need to be stripped off *)
WHILE RIGHT(TRIME,1) = ' ' DO
	TRIME := DELETE(TRIME,1,LEN(TRIME));
END_WHILE;


(* revision histroy
hm	28. mar. 2008	rev 1.0
	original release

*)
END_FUNCTION

(* POU Time&Date/CALENDAR_CALC, ST *)
FUNCTION_BLOCK CALENDAR_CALC
VAR_INPUT
	SPE : BOOL;
	H : REAL := -0.83333333333;
END_VAR
VAR_IN_OUT
	XCAL : CALENDAR;
	HOLIDAYS : ARRAY[0..29] OF HOLIDAY_DATA;
END_VAR
VAR
	last : DT;
	last_day : DINT;
	holy : HOLIDAY;
	sun : SUN_TIME;
	last_hour: INT;
	utod: TOD;
	pos : SUN_POS;
	plast: DT;
END_VAR
VAR_TEMP
	dtemp : DINT;
	tmp : INT;
END_VAR


(*
version 1.6	6. apr. 2011
programmer 	hugo
tested by		oscat

calendar_calc liest die weltzeit .UTC aus einer CALENDAR Struktur und berechnet die restlichen Werte der Struktur.
calendar_calc stellt sicher das die Werte fortlaufend aktualisiert werden und dabei funktionen nur dann aufgerufen werden wenn dies nötig ist.
calendar_calc will calculate sun position data when SPE = TRUE;

*)
IF xcal.UTC <> last THEN
	(* run once per second *)
	(* update utc last calculated  *)
	last := XCAL.UTC;
	utod := DT_TO_TOD(xcal.UTC);

	(* calculate ltc from utc *)
	XCAL.LDT := UTC_TO_LTIME(XCAL.UTC, XCAL.DST_EN, XCAL.OFFSET);
	XCAL.LDATE := DT_TO_DATE(XCAL.LDT);
	XCAL.LTOD := DT_TO_TOD(XCAL.LDT);
	dtemp := DAY_OF_DATE(XCAL.LDATE);
	xcal.night := XCAL.LTOD < XCAL.SUN_RISE OR XCAL.LTOD > XCAL.SUN_SET;

	(* run once per hour *)
	tmp := HOUR(xcal.LTOD);
	IF  tmp <> last_hour THEN
		XCAL.DST_ON := DST(XCAL.UTC) AND xcal.DST_EN;
		last_hour := tmp;
	END_IF;

	(* run once per day *)
	IF dtemp <> last_day THEN
		last_day := dtemp;
		(* a new day has started, recalculate daily events *)
		XCAL.YEAR := YEAR_OF_DATE(XCAL.LDATE);
		XCAL.MONTH := MONTH_OF_DATE(XCAL.LDATE);
		XCAL.DAY := DAY_OF_MONTH(XCAL.LDATE);
		XCAL.WEEKDAY := DAY_OF_WEEK(XCAL.LDATE);
		HOLY(date_in := XCAL.LDATE, LANGU := xcal.LANGUAGE, HOLIDAYS := HOLIDAYS);
		XCAL.HOLIDAY := HOLY.Y;
		XCAL.HOLY_NAME := HOLY.NAME;
		sun(latitude := XCAL.LATITUDE, longitude := xcal.LONGITUDE, utc := DT_TO_DATE(xcal.UTC), H := H);
		XCAL.SUN_RISE := DINT_TO_TOD(TOD_TO_DINT(sun.sun_rise) + XCAL.OFFSET * 60000 + SEL(XCAL.DST_ON,DINT#0,3600000));
		XCAL.SUN_SET := DINT_TO_TOD(TOD_TO_DINT(sun.sun_set) + XCAL.OFFSET * 60000 + SEL(XCAL.DST_ON,DINT#0,3600000));
		XCAL.SUN_MIDDAY := DINT_TO_TOD(TOD_TO_DINT(sun.MIDDAY) + XCAL.OFFSET * 60000 + SEL(XCAL.DST_ON,DINT#0,3600000));
		XCAL.SUN_HEIGTH := sun.sun_declination;
		XCAL.WORK_WEEK := WORK_WEEK(XCAL.LDATE);
	END_IF;

	(* calculate the suns position every 10 seconds when SPE = TRUE *)
	IF SPE AND xcal.UTC -  plast >= t#25s THEN
		plast := last;
		pos(latitude := xcal.LATITUDE, longitude := xcal.LONGITUDE, utc := xcal.UTC);
		xcal.SUN_HOR := pos.B;
		xcal.SUN_VER := pos.HR;
	END_IF;
END_IF;



(* revision history

hm 23. oct. 2008	rev 1.0
	original version

hm	8. feb. 2009	rev 1.1
	night was calculated wrong
	added sun position data

hm	10. mar. 2009	rev 1.2
	added work_week, sun_midday, sun_heigth
	sun_position will only be calculated evey 25 seconds
	dst will only become true when dst_en = true

hm	23. jan 2010	rev 1.3
	sun_rise, sun_set and sun_midday are now calculated in local time

hm	18. jan. 2011	rev 1.4
	added input holidays to specify local holidays
	changed call for function sun_time

hm	2. feb. 2011	rev 1.5
	added input H to specify twilight

hm	6. apr. 2011	rev 1.6
	night was calculated wrong
*)
END_FUNCTION_BLOCK

(* POU Time&Date/HOLIDAY, ST *)
FUNCTION_BLOCK HOLIDAY
VAR_INPUT
	DATE_IN : DATE;
	LANGU : INT;
	FRIDAY : BOOL;
	SATURDAY : BOOL;
	SUNDAY : BOOL;
END_VAR
VAR_IN_OUT
	HOLIDAYS : ARRAY[0..29] OF HOLIDAY_DATA;
END_VAR
VAR CONSTANT
	SIZE : INT := 29;
END_VAR
VAR_OUTPUT
	Y : BOOL;
	NAME : STRING(30);
END_VAR
VAR
	last_active : DATE;
	ostern: DATE;
	i: INT;
	jahr: INT;
	x_date: DATE;
	lx: INT;
	wdx: INT;
END_VAR

(*
version 2.0	18. jans 2011
programmer 	hugo
tested by		tobias

holiday calculates if a given day is a holiday and displays the name of the holiday as string as well as a boolean flag to indicate a holiday.
the holidays are specified in the country setup under global constants.
a holiday can be of fixed date for example new years day on january 1st.
a holiday can have a fixed offset from easter sunday as for most church holidays.
a holiday can be a specific weekday before a fixed date, for example buss und bettag is the last wednesday before nov 23rd.
with a simple f_use flag any specific holiday can be turned on or off if needed.

please check the manual for examples of holiday definitions
*)
(* for performance reasons only activate once a day *)
IF last_active = date_in THEN RETURN; END_IF;
last_active := DATE_IN;

(* determine language *)
IF LANGU = 0 THEN
	lx := language.DEFAULT;
ELSE
	lx := MIN(language.LMAX, LANGU);
END_IF;

(* berechnung von ostern für das aktuelle jahr *)
jahr := YEAR_OF_DATE(date_in);
ostern := EASTER(jahr);
wdx := DAY_OF_WEEK(DATE_IN);
Y := FALSE;

(* check for holidays *)
FOR i := 0 TO size DO
	x_date := SET_DATE(jahr, HOLIDAYS[i].MONTH , HOLIDAYS[i].DAY);
	IF HOLIDAYS[i].USE = 1 AND HOLIDAYS[i].MONTH > 0 THEN
		(* check for fixed date holiday *)
		IF x_date = date_in THEN
			Y := TRUE;
			NAME := HOLIDAYS[i].NAME;
			RETURN;
		END_IF;
	ELSIF HOLIDAYS[i].USE = 1 AND HOLIDAYS[i].MONTH = 0 THEN
		(* check for holiday in reference to easter *)
		IF DATE_ADD(ostern, HOLIDAYS[i].DAY ,0,0,0) = date_in THEN
			Y := TRUE;
			NAME := HOLIDAYS[i].NAME;
			RETURN;
		END_IF;
	ELSIF HOLIDAYS[i].USE < 0 THEN
		(* check for holiday on a weekday before date *)
		IF DAY_OF_WEEK(date_in) = ABS(HOLIDAYS[i].USE) AND date_in < x_date AND date_in >= DATE_ADD(x_date,-7,0,0,0) THEN
			Y := TRUE;
			NAME := HOLIDAYS[i].NAME;
			RETURN;
		END_IF;
	END_IF;
END_FOR;

(* check array if today is weekend *)
IF NOT Y AND (wdx = 5 AND FRIDAY OR wdx = 6 AND SATURDAY OR wdx = 7 AND SUNDAY) THEN
	Y := TRUE;
	NAME := LANGUAGE.WEEKDAYS[LOCATION.LANGUAGE[lx],wdx];
ELSE
	NAME := '';
END_IF;


(*
Neujahrstag 	1. Januar 	• 	• 	• 	• 	• 	• 	• 	• 	• 	• 	• 	• 	• 	• 	• 	•
Heilige Drei Könige 	6. Januar 	• 	• 												• 		
Karfreitag 	Ostersonntag - 2d 	• 	• 	• 	• 	• 	• 	• 	• 	• 	• 	• 	• 	• 	• 	• 	•
Ostersonntag 	siehe Osterdatum 				(•) 												
Ostermontag 	Ostersonntag + 1d 	• 	• 	• 	• 	• 	• 	• 	• 	• 	• 	• 	• 	• 	• 	• 	•
Tag der Arbeit 	1. Mai 	• 	• 	• 	• 	• 	• 	• 	• 	• 	• 	• 	• 	• 	• 	• 	•
Christi Himmelfahrt 	Ostersonntag + 39d 	• 	• 	• 	• 	• 	• 	• 	• 	• 	• 	• 	• 	• 	• 	• 	•
Pfingstsonntag 	Ostersonntag + 49d 				(•) 												
Pfingstmontag 	Ostersonntag + 50d 	• 	• 	• 	• 	• 	• 	• 	• 	• 	• 	• 	• 	• 	• 	• 	•
Fronleichnam 	Ostersonntag + 60d 	• 	• 					• 			• 	• 	• 	1) 			2)
Augsburger Friedensfest 	8. August 		(3) 														
Mariä Himmelfahrt 	15. August 		(5) 										• 				
Tag der Deutschen Einheit 	3. Oktober 6) 	• 	• 	• 	• 	• 	• 	• 	• 	• 	• 	• 	• 	• 	• 	• 	•
Reformationstag 	31. Oktober 				• 				• 					• 	• 		•
Allerheiligen 	1. November 	• 	• 								• 	• 	• 				
Buß- und Bettag 4) 	Mittwoch vor dem 23.11. 			7 										• 			
1. Weihnachtstag 	25. Dezember 	• 	• 	• 	• 	• 	• 	• 	• 	• 	• 	• 	• 	• 	• 	• 	•
2. Weihnachtstag 	26. Dezember 	• 	• 	• 	• 	• 	• 	• 	• 	• 	• 	• 	• 	• 	• 	• 	•
*)



(* revision history
hm 	27. feb. 2007	rev 1.1
	deleted unused variable init

hm	31. oct. 2007	rev 1.2
	changed holiday definition from constant to input constant to allow easier changes by user without recompilation of the lib

hm 	24. nov. 2007	rev 1.3
	changes F_use of  Buß_und_Bettag to 0 because this is no official holiday

hm	7. apr. 2008	rev 1.4
	improved performance

hm	7. oct. 2008	rev 1.5
	changed code to use setup data from global constants
	changed length of output NAME from 20 to 30
	holiday will now also be indicated on a weekend
	changed function year to year_of_date
	changed function weekday to day_of_week

hm	21. oct. 2008	rev 1.6
	using location constants

hm	18. jan 2011	rev 2.0
	using user specified array for holidays

*)
END_FUNCTION_BLOCK

(* POU Time&Date/EASTER, ST *)
FUNCTION EASTER : DATE
VAR_INPUT
	year : INT;
END_VAR
VAR
	b,c: INT;
	oday: INT;
END_VAR

(*
version 1.3	7. apr. 2008
programmer 	hugo
tested by	tobias

easter calculates the day of easter sunday for a given year.
most other catholic holidays are calculated in reference to easter sunday.

*)
b := (204 - 11 * (YEAR MOD 19)) MOD 30;
IF b > 27 THEN b := b - 1; END_IF;
c := (year + SHR(year,2) + b - 13) MOD 7;
oday := 28 + b - c;
IF oday > 33 THEN
	EASTER := SET_DATE(year, 4, oday - 31);
ELSE
	EASTER := SET_DATE(year, 3, oday);
END_IF;




(* alternativer algorithmus ueber das pasah fest
execution time roughly 200us
Der sog. Passah-Vollmond wird berechnet, in dem das Jahr durch 19 ge-
teilt wird und der Rest mit der folgenden Tabelle verglichen wird:
 
    0: Apr 14       5: Apr 18      10: Mrz 25      15: Mrz 30
    1: Apr 03       6: Apr 08      11: Apr 13      16: Apr 17
    2: Mrz 23       7: Mrz 28      12: Apr 02      17: Apr 07
    3: Apr 11       8: Apr 16      13: Mrz 22      18: Mrz 27
    4: Mrz 31       9: Apr 05      14: Apr 10
 
Faellt dieses Datum auf einen Sonntag, ist Ostern der naechste Sonntag!
 
Beispiel: 1992 MOD 19 = 16, daraus folgt 17.04., der naechste Sonntag
          ist dann der 19. April (Ostersonntag)
*)


(* this algorithm is 180 us
a := year MOD 19;
b := year / 100;
c := year MOD 100;
d := b / 4;
e := b MOD 4;
f := (b + 8) / 25;
g := (b - f + 1) / 3;
h := (19 * a + b - d -g + 15) MOD 30;
i := C / 4;
k := c MOD 4;
l := (32 + 2*e + 2*i - h - k) MOD 7;
m := (a + 11 * h + 22 * l) / 451;
x := h + l - 7 * m + 114;
n := X / 31;
o := x MOD 31 + 1;

easter := set_Date(year,n,o);
*)
(*
Im Magazin "Nature" vom 20. April 1876 veröffentlichte ein anonymer Autor eine Tabelle mit Regeln zur Berechnung des (Gregorianischen) Ostersonntages des Jahres J. In Formeln ausgedrückt erhält man das Folgende:
a	=	J mod 19
b	=	int(J / 100)
c	=	J mod 100
d	=	int(b / 4)
e	=	b mod 4
f	=	int((b + 8) / 25)
g	=	int((b - f + 1) / 3
h	=	(19 · a + b - d - g + 15) mod 30
i	=	int(c / 4)
k	=	c mod 4
l	=	(32 + 2 · e + 2 · i - h - k) mod 7
m	=	int((a + 11 · h + 22 · l) / 451)
n	=	int((h + l - 7 · m + 114) / 31)
o	=	(h + l - 7 · m + 114) mod 31

n ist hierbei die Nummer des Monats, o + 1 die Nummer des Tages auf welchen der Ostersonntag im Jahr J fällt. Dieser Algorithmus kommt ohne Hilfszahlen aus.

*)

(* revision history
hm	27. dec 2006	rev 1.0
	original version

hm	15. dec 2007	rev 1.1
	modified code for better performance

hm	3. feb 2008		rev 1.2
	modified code for better performance

hm	7. apr. 2008	rev 1.3
	improved performance
*)
END_FUNCTION

(* POU Time&Date/DATE_ADD, ST *)
FUNCTION DATE_ADD : DATE
VAR_INPUT
	IDATE : DATE;
	D : INT;
	W : INT;
	M : INT;
	Y : INT;
END_VAR
VAR
	mo: INT;
	yr : INT;
	dm: INT;
END_VAR


(*
version 1.8		22. mar. 2011
programmer 	hugo
tested by		oscat

date_add adds days, weeks, month or years to a date.
negative inputs are allowed for subtraction.

*)
DATE_ADD := UDINT_TO_DATE(DATE_TO_UDINT(IDATE) + INT_TO_UDINT(D + W * 7) * UDINT#86400);
yr := Y + YEAR_OF_DATE(DATE_ADD);
mo := M + MONTH_OF_DATE(DATE_ADD);
dm := DAY_OF_MONTH(DATE_ADD);
WHILE mo > 12 DO
	mo := mo - 12;
	yr := yr + 1;
END_WHILE;
WHILE mo < 1 DO
	mo := mo + 12;
	yr := yr - 1;
END_WHILE;
DATE_ADD := SET_DATE(yr, mo, dm);


(* revision history

hm 27.12.2006	rev 1.0
	nrw module

hm 12.4.2007		rev 1.1
	corrected an error while date would be incorrect when year  = 0

hm	1.11.2007		rev 1.2
	added int_to_dword stetements to avoid possible overrun with möller ecp4

hm	22. mar. 2008	rev 1.3
	fixed some bugs when month was negative

hm	7. oct. 2008	rev 1.4
	changed function year to year_of_date
	changed function month to month_of_date

hm	29. mar. 2009	rev 1.5
	improved performance

hm	27. jan. 2011	rev 1.6
	faster code

hm	2. feb. 2011		rev 1.7
	fixed an error, weeks not calculated

hm	22. mar. 2011	rev 1.8
	fixed an error in formula
*)
END_FUNCTION

(* POU Time&Date/SUN_TIME, ST *)
FUNCTION_BLOCK SUN_TIME
VAR_INPUT
	LATITUDE : REAL;				(* latitude of geographical position  *)
	LONGITUDE : REAL;				(* longitude of geographical position  *)
	UTC : DATE;						(*	world time	*)
	H : REAL := -0.83333333333;	(* heighth above horizon for sunrise *)
END_VAR
VAR_OUTPUT
	MIDDAY : TOD;			(*	astrological midday in hours when sun stands at south direction	*)
	SUN_RISE : TOD;				(*	sun rise for current day in local time *)
	SUN_SET : TOD;				(*	sun set for current day in local time *)
	SUN_DECLINATION : REAL;		(*	sun declination above horizon at midday in degrees	*)
END_VAR
VAR
	dk: REAL;						(* sun declination at midday *)
	delta: TIME;					(* delta from midday for sunrise and sunset  *)
	b: REAL;
END_VAR

(*
version 1.7	25. jan. 2011
programmer 	hugo
tested by	tobias

this FUNCTION block calculates the sun rise, sun set, sun offset at midday sun declination for a given date 
for performance reasons the algorithm has been simplified and is accurate within a few minutes only 
the times are calculated in utc and have to be corrected for the given time zone
this correction is not done within sun_time because it would be a problem on days where dst is enabled or disabled

*)
B := latitude * 0.0174532925199433;
MIDDAY := SUN_MIDDAY(longitude, utc);
DK := 0.40954 * SIN(0.0172 * (INT_TO_REAL(DAY_OF_YEAR(utc)) - 79.35));
sun_declination := DEG(DK);
IF sun_declination > 180.0 THEN sun_declination := sun_declination - 360.0; END_IF;
sun_declination := 90.0 - LATITUDE + sun_declination;
delta := HOUR_TO_TIME(ACOS((SIN(RAD(H)) - SIN(B) * SIN(DK)) / (COS(B) * COS(DK))) * 3.819718632);
sun_rise := MIDDAY - delta;
sun_set := MIDDAY + delta;

(* revision history

rev 1.1	hm	20.1.2007
	deleted unused variables sun_riseR and sun_setR

rev 1.2 hm 17.4.2007
	corrected error while sun:midday would not be corrected for longitude.

rev 1.3	hm	6. jan 2008
	performance improvements

rev	1.4 hm	17. jan 2008
	calculation is now only performed once a day

hm	10. mar. 2009	rev 1.5
	improved performance
	calculation will be performed on every call to allow movong installations

hm	26. jul 2009	rev 1.6
	fixed a problem with wrong midday calculation

hm	25. jan. 2011	rev 1.7
	using function sun_midday
	corrected angle of sun_declination
	added input H
*)
END_FUNCTION_BLOCK

(* POU Time&Date/SUN_MIDDAY, ST *)
FUNCTION SUN_MIDDAY : TOD
VAR_INPUT
	LON : REAL;
	UTC : DATE;
END_VAR
VAR
	T : REAL;
	OFFSET : REAL;
END_VAR

(*
version 1.0	26. jan. 2011
programmer 	hugo
tested by	oscat

this FUNCTION calculates the time when the sun stand exactly south of a given location.

*)
T := INT_TO_REAL(DAY_OF_YEAR(utc));
OFFSET := -0.1752 * SIN(0.033430 * T + 0.5474) - 0.1340 * SIN(0.018234 * T - 0.1939);
SUN_MIDDAY := HOUR_TO_TOD(12.0 - OFFSET - lon * 0.0666666666666);


(* revision history

hm	26. jan. 2011	rev 1.0
	initial release

*)
END_FUNCTION

(* POU Time&Date/HOUR_TO_TOD, ST *)
FUNCTION HOUR_TO_TOD : TOD
VAR_INPUT
	IN : REAL;
END_VAR


(*
version 1.2	24. feb 2009
programmer 	hugo
tested by		tobias

converts an amount of hours in real to time of day TOD.

*)
HOUR_TO_TOD := DWORD_TO_TOD(REAL_TO_DWORD(IN * 3600000));


(* revision history
hm	4. aug. 2006	rev 1.0
	original version

hm	14. mar. 2008	rev 1.1
	rounded the input after the last digit

hm	24. feb. 2009	rev 1.2
	changed input to IN
*)
END_FUNCTION

(* POU Time&Date/HOUR_TO_TIME, ST *)
FUNCTION HOUR_TO_TIME : TIME
VAR_INPUT
	IN : REAL;
END_VAR


(*
version 1.2	24. feb. 2009
programmer 	hugo
tested by		tobias

converts an amount of hours in real to time

*)
HOUR_TO_TIME := DWORD_TO_TIME(REAL_TO_DWORD(IN * 3600000));


(* revision history
hm		4. aug 2006	rev 1.0
	original version

hm	14. mar. 2008	rev 1.1
	rounded the input after the last digit

hm	24. feb. 2009	rev 1.2
	changed input to IN
*)
END_FUNCTION

(* POU Time&Date/SUN_POS, ST *)
FUNCTION_BLOCK SUN_POS
VAR_INPUT
	latitude : REAL;				(* latitude of geographical position  *)
	longitude : REAL;				(* longitude of geographical position  *)
	utc : DT;						(*	world time				*)
END_VAR
VAR_OUTPUT
	B: REAL;
	H : REAL;
	HR: REAL;
END_VAR
VAR_TEMP
	g: REAL;
	a: REAL;
	d: REAL;
	t1: REAL;
	n: REAL;
	e: REAL;
	c: REAL;
	tau: REAL;
	sin_d: REAL;
	rlat: REAL;
	sin_lat: REAL;
	cos_lat: REAL;
	cos_tau: REAL;
	cos_d: REAL;
END_VAR

(*
version 2.1	7. mar. 2009
programmer 	hugo
tested by		oscat

this FUNCTION block calculates the sun position for a given date and time.
the times are calculated in utc and have to be corrected for the given time zone.
B is the angle from north and HR is the highth in degrees.

*)
(* n is the julian date and the number of days since 1.1.2000-12:00 midday *)
(* be careful for step7 date startes 1.1.1990 instead of 1.1.1970 *)
(* for step7 this line must change *)
n := DWORD_TO_REAL(DT_TO_DWORD(UTC) - 946728000) * 0.000011574074074074;
g :=MODR(6.240040768 + 0.01720197 * n, math.PI2);
d := MODR(4.89495042 + 0.017202792 * n, math.PI2) + 0.033423055 * SIN(g) + 0.000349066 * SIN(2.0*g);
e := 0.409087723 - 0.000000006981317008 * n;
cos_d := COS(d);
sin_d := SIN(d);
a := ATAN(COS(e) * sin_d / cos_d);
IF cos_d < 0.0 THEN a := a + math.PI; END_IF;
c := ASIN(SIN(e) * sin_d);

(* also here we must be very careful utc is from 1.1.1970 for step7 the formula must change *)
tau := RAD(MODR(6.697376 + (n - 0.25) * 0.0657098245037645 + DWORD_TO_REAL(TOD_TO_DWORD(DT_TO_TOD(utc))) * 0.0000002785383333, 24.0) * 15.0 + longitude) - a;
rlat := RAD(latitude);
sin_lat := SIN(rlat);
cos_lat := COS(rlat);
cos_tau := COS(tau);
t1 := cos_tau * sin_lat - TAN(c) * cos_lat;
B := ATAN(SIN(tau) / t1);
IF t1< 0.0 THEN B := B + math.PI2; ELSE B := B + math.PI; END_IF;
B := DEG(MODR(B, math.PI2));
h := DEG(ASIN(COS(C) * cos_tau * cos_lat +SIN(c) * sin_lat));
IF h > 180.0 THEN h := h - 360.0; END_IF;
(* consider refraction *)
HR := h + REFRACTION(h);


(* revision history
hm	1. feb 2007	rev 1.0
	original version

hm	6. jan 2008	rev 1.1
	performance improvements

hm	18. jan 2008	rev 1.2
	further performance improvements
	only calculate once every 10 seconds

hm	16. mar. 2008	rev 1.3
	added type conversion to avoid warnings under codesys 3.0

hm	30. jun. 2008	rev 1.4
	added type conversions to avoid warnings under codesys 3.0

hm	18. oct. 2008	rev 1.5
	using math constants

hm	17. dec. 2008	rev 1.6
	angles below horizon are displayed in negative degrees

hm	27. feb. 2009	rev 2.0
	new code with better accuracy

hm	7. mar. 2009	rev 2.1
	refraction is added after angle normalization
	deleted 10 second lockout
	added output for astronomical heigth h
*)
END_FUNCTION_BLOCK

(* POU Time&Date/REFRACTION, ST *)
FUNCTION REFRACTION : REAL
VAR_INPUT
	ELEV : REAL;
END_VAR


(*
version 1.1	7. mar. 2009
programmer 	hugo
tested by		oscat

REFRACTION calculates the atmospheric refraction in degrees.
the input angle goes from 0 at the hirizon to 90 at midday.

*)
elev := LIMIT(-1.9, elev, 80.0);
REFRACTION := 0.0174532925199433 / TAN(0.0174532925199433 * (ELEV + 10.3 / (ELEV + 5.11)));


(* revision histroy
hm	14. jul. 2008	rev 1.0
	original release

hm	7. mar. 2009	rev 1.1
	using new formula

*)	
END_FUNCTION

(* POU Time&Date/UTC_TO_LTIME, ST *)
FUNCTION UTC_TO_LTIME : DT
VAR_INPUT
	UTC : DT;
	DST_ENABLE : BOOL;
	TIME_ZONE_OFFSET : INT;
END_VAR
VAR
	tmp: INT;
END_VAR

(*

version 1.9	27. feb. 2009
programmer 	oscat
tested by		oscat

ltime is a real time clock that uses the system rtc as utc time and calculates and given time zone.
the utc time is supplied on the input UTC.
according to the input variable time_zone_offset when the input dst_enable is true,
the dst on and off times are calculated by a formula for any given year and the time is advanced and reset by one hour
at 02:00 and 03:00 for the last sunday of march and last sunday of october.
the code is high performance and the rtc counts every second.
if more then one time zone is needed by the systen the clock can be started many times by placing more then one function block.

 
